KUKA KRL program: EPS_2_251491_MH04A_A_20251118025158.src

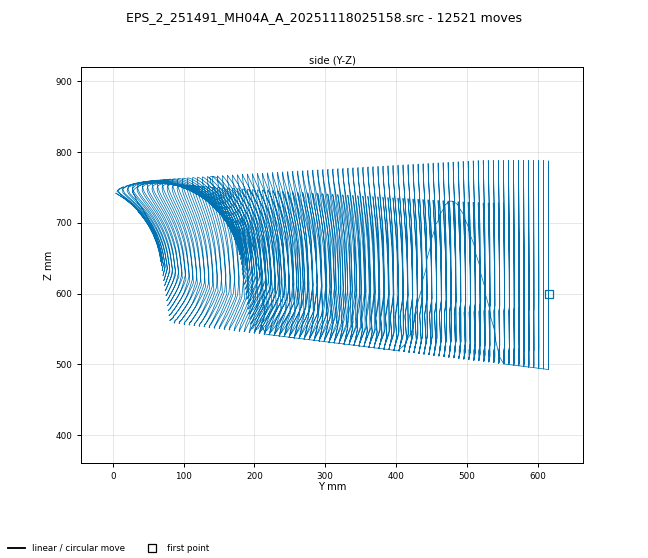
[picture p0: tool path of EPS_2_251491_MH04A_A_20251118025158.src, 12521 of 12523 moves have a stored position in this frame; points joined in program order, loops and branches not executed]
&ACCESS RVP
&REL 4
&COMMENT QRS 19112012
&PARAM EDITMASK = *
DEF PART()
EXT BAS (BAS_COMMAND :IN,REAL :IN )
INT I
BAS (#INITMOV,0 )

;KUKA QRS Post kuka4.cps  Date:22-06-2017 !

File_ID=2918

QRS_PRE_INIT()

;Init var - Until changes are made in qrs_pre_init
Outlet_Square_prg=0
Inlet_1_Square_prg=0
Inlet_2_Square_prg=0
Inlet_3_Square_prg=0
Inlet_4_Square_prg=0
Inlet_5_Square_prg=0

Outlet_1={X 0.000, Y 519.160, Z 687.500, B 0.000, E1 0.000 }
Inlet_1={X 0.000, Y 523.440, Z 627.500, B 0.000, E1 142.000 }
Outlet_1_type=201
Inlet_1_type=201
;QRS#1=Sidecore dimensions
;QRS#2=200-8" PVC SDR 35
;QRS#3=200-8" PVC SDR 35
;QRS#4=
;QRS#5=
;QRS#6=
;QRS#7=
;QRS#8=
;QRS#9=12-08 PSX
;QRS#10=12-08 PSX
;QRS#11=
;QRS#12=
;QRS#13=
;QRS#14=
;QRS#15=
;QRS#16=1220x127x1067 3,5'
;QRS#17=EPS Height
;QRS#18=788
;QRS#19=*
;QRS#20= UPDATED VERSION 22-06-2017
;QRS#21=*
Outlet_Square=0100
Inlet_1_Square=0100
Inlet_2_Square=0
Inlet_3_Square=0
Inlet_4_Square=0
Inlet_5_Square=0
Mill_Square=1
Outlet_Square_Prg=204
Inlet_1_Square_prg=204

QRS_INIT()

$ADVANCE=5

; T1
PTP {E1 173.594,E2 173.594}
PTP {X 0,Y 615.502,A -85,B 0,C 180,E1 173.594,E2 173.594,E3 0,E4 0,E5 0,E6 0}
QRS_SPEED_INIT()
LIN {X 0,Y 615.502,Z 600,A -85,B 0,C 180,E1 173.594,E2 173.594,E3 0,E4 0,E5 0,E6 0} C_VEL
LIN {X 0,Y 615.502,Z 502.864,A -85,B 0,C 180,E1 173.594,E2 173.594} C_VEL
LIN {X 0,Y 615.502,Z 494.687,A -85,B 0,C 180,E1 173.594,E2 173.594} C_VEL
LIN {X 0,Y 615.49,Z 492.687,A -85,B 0,C 180,E1 173.408,E2 173.408} C_VEL
LIN {X 0,Y 615.493,Z 492.697,A -85,B 0,C 180,E1 170.802,E2 170.802} C_VEL
LIN {X 0,Y 615.479,Z 492.685,A -85,B 0,C 180,E1 168.139,E2 168.139} C_VEL
LIN {X 0,Y 615.488,Z 492.686,A -85,B 0,C 180,E1 165.451,E2 165.451} C_VEL
LIN {X 0,Y 615.494,Z 492.696,A -85,B 0,C 180,E1 162.73,E2 162.73} C_VEL
LIN {X 0,Y 615.477,Z 492.684,A -85,B 0,C 180,E1 159.967,E2 159.967} C_VEL
LIN {X 0,Y 615.486,Z 492.692,A -85,B 0,C 180,E1 157.156,E2 157.156} C_VEL
LIN {X 0,Y 615.493,Z 492.685,A -85,B 0,C 180,E1 154.285,E2 154.285} C_VEL
LIN {X 0,Y 615.486,Z 492.686,A -85,B 0,C 180,E1 151.342,E2 151.342} C_VEL
LIN {X 0,Y 615.492,Z 492.697,A -85,B 0,C 180,E1 148.911,E2 148.911} C_VEL
LIN {X 0,Y 615.479,Z 492.684,A -85,B 0,C 180,E1 145.978,E2 145.978} C_VEL
LIN {X 0,Y 615.49,Z 492.767,A -85,B 0,C 180,E1 145.297,E2 145.297} C_VEL
LIN {X 0,Y 615.493,Z 508.915,A -85,B 0,C 180,E1 142.373,E2 142.373} C_VEL
LIN {X 0,Y 615.476,Z 517.644,A -85,B 0,C 180,E1 140.809,E2 140.809} C_VEL
LIN {X 0,Y 615.481,Z 623.163,A -85,B 0,C 180,E1 139.556,E2 139.556} C_VEL
LIN {X 0,Y 615.482,Z 636.415,A -85,B 0,C 180,E1 139.271,E2 139.271} C_VEL
LIN {X 0,Y 615.49,Z 649.214,A -85,B 0,C 180,E1 138.857,E2 138.857} C_VEL
LIN {X 0,Y 615.497,Z 660.234,A -85,B 0,C 180,E1 138.376,E2 138.376} C_VEL
LIN {X 0,Y 615.48,Z 670.961,A -85,B 0,C 180,E1 137.783,E2 137.783} C_VEL
LIN {X 0,Y 615.495,Z 681.65,A -85,B 0,C 180,E1 137.038,E2 137.038} C_VEL
LIN {X 0,Y 615.496,Z 691.498,A -85,B 0,C 180,E1 136.19,E2 136.19} C_VEL
LIN {X 0,Y 615.494,Z 700.206,A -85,B 0,C 180,E1 135.263,E2 135.263} C_VEL
LIN {X 0,Y 615.495,Z 707.231,A -85,B 0,C 180,E1 134.343,E2 134.343} C_VEL
LIN {X 0,Y 615.499,Z 713.951,A -85,B 0,C 180,E1 133.242,E2 133.242} C_VEL
LIN {X 0,Y 615.498,Z 719.396,A -85,B 0,C 180,E1 132.082,E2 132.082} C_VEL
LIN {X 0,Y 615.495,Z 722.82,A -85,B 0,C 180,E1 131.096,E2 131.096} C_VEL
LIN {X 0,Y 615.498,Z 725.29,A -85,B 0,C 180,E1 130.091,E2 130.091} C_VEL
LIN {X 0,Y 615.491,Z 726.968,A -85,B 0,C 180,E1 128.903,E2 128.903} C_VEL
LIN {X 0,Y 615.493,Z 727.381,A -85,B 0,C 180,E1 128.013,E2 128.013} C_VEL
LIN {X 0,Y 615.492,Z 726.916,A -85,B 0,C 180,E1 126.938,E2 126.938} C_VEL
LIN {X 0,Y 615.496,Z 725.326,A -85,B 0,C 180,E1 125.836,E2 125.836} C_VEL
LIN {X 0,Y 615.494,Z 722.463,A -85,B 0,C 180,E1 124.702,E2 124.702} C_VEL
LIN {X 0,Y 615.494,Z 718.151,A -85,B 0,C 180,E1 123.536,E2 123.536} C_VEL
LIN {X 0,Y 615.496,Z 712.793,A -85,B 0,C 180,E1 122.456,E2 122.456} C_VEL
LIN {X 0,Y 615.496,Z 705.972,A -85,B 0,C 180,E1 121.385,E2 121.385} C_VEL
LIN {X 0,Y 615.497,Z 697.582,A -85,B 0,C 180,E1 120.348,E2 120.348} C_VEL
LIN {X 0,Y 615.498,Z 689.18,A -85,B 0,C 180,E1 119.503,E2 119.503} C_VEL
LIN {X 0,Y 615.495,Z 678.79,A -85,B 0,C 180,E1 118.657,E2 118.657} C_VEL
LIN {X 0,Y 615.485,Z 667.368,A -85,B 0,C 180,E1 117.914,E2 117.914} C_VEL
LIN {X 0,Y 615.487,Z 655.583,A -85,B 0,C 180,E1 117.314,E2 117.314} C_VEL
LIN {X 0,Y 615.479,Z 642.588,A -85,B 0,C 180,E1 116.821,E2 116.821} C_VEL
LIN {X 0,Y 615.479,Z 629.925,A -85,B 0,C 180,E1 116.481,E2 116.481} C_VEL
LIN {X 0,Y 615.491,Z 616.108,A -85,B 0,C 180,E1 116.261,E2 116.261} C_VEL
LIN {X 0,Y 615.49,Z 517.628,A -85,B 0,C 180,E1 115.099,E2 115.099} C_VEL
LIN {X 0,Y 615.496,Z 501.148,A -85,B 0,C 180,E1 112.136,E2 112.136} C_VEL
LIN {X 0,Y 615.476,Z 492.688,A -85,B 0,C 180,E1 110.577,E2 110.577} C_VEL
LIN {X 0,Y 615.486,Z 492.683,A -85,B 0,C 180,E1 107.957,E2 107.957} C_VEL
LIN {X 0,Y 615.489,Z 492.699,A -85,B 0,C 180,E1 105.226,E2 105.226} C_VEL
LIN {X 0,Y 615.477,Z 492.688,A -85,B 0,C 180,E1 102.53,E2 102.53} C_VEL
LIN {X 0,Y 615.486,Z 492.683,A -85,B 0,C 180,E1 99.862,E2 99.862} C_VEL
LIN {X 0,Y 615.491,Z 492.698,A -85,B 0,C 180,E1 97.215,E2 97.215} C_VEL
LIN {X 0,Y 615.477,Z 492.689,A -85,B 0,C 180,E1 94.585,E2 94.585} C_VEL
LIN {X 0,Y 615.496,Z 492.68,A -85,B 0,C 180,E1 91.963,E2 91.963} C_VEL
LIN {X 0,Y 615.484,Z 492.694,A -85,B 0,C 180,E1 89.346,E2 89.346} C_VEL
LIN {X 0,Y 615.482,Z 492.692,A -85,B 0,C 180,E1 86.727,E2 86.727} C_VEL
LIN {X 0,Y 615.488,Z 492.681,A -85,B 0,C 180,E1 84.102,E2 84.102} C_VEL
LIN {X 0,Y 615.479,Z 492.691,A -85,B 0,C 180,E1 81.463,E2 81.463} C_VEL
LIN {X 0,Y 615.489,Z 492.694,A -85,B 0,C 180,E1 78.807,E2 78.807} C_VEL
LIN {X 0,Y 615.485,Z 492.682,A -85,B 0,C 180,E1 76.067,E2 76.067} C_VEL
LIN {X 0,Y 615.482,Z 492.691,A -85,B 0,C 180,E1 73.414,E2 73.414} C_VEL
LIN {X 0,Y 615.483,Z 492.691,A -85,B 0,C 180,E1 70.662,E2 70.662} C_VEL
LIN {X 0,Y 615.495,Z 492.68,A -85,B 0,C 180,E1 67.864,E2 67.864} C_VEL
LIN {X 0,Y 615.495,Z 492.701,A -85,B 0,C 180,E1 65.009,E2 65.009} C_VEL
LIN {X 0,Y 615.483,Z 492.683,A -85,B 0,C 180,E1 62.085,E2 62.085} C_VEL
LIN {X 0,Y 615.499,Z 492.679,A -85,B 0,C 180,E1 59.841,E2 59.841} C_VEL
LIN {X 0,Y 615.485,Z 492.686,A -85,B 0,C 180,E1 57.543,E2 57.543} C_VEL
LIN {X 0,Y 615.482,Z 492.696,A -85,B 0,C 180,E1 55.186,E2 55.186} C_VEL
LIN {X 0,Y 615.492,Z 492.694,A -85,B 0,C 180,E1 52.759,E2 52.759} C_VEL
LIN {X 0,Y 615.489,Z 492.681,A -85,B 0,C 180,E1 49.91,E2 49.91} C_VEL
LIN {X 0,Y 615.493,Z 492.701,A -85,B 0,C 180,E1 46.951,E2 46.951} C_VEL
LIN {X 0,Y 615.482,Z 492.683,A -85,B 0,C 180,E1 43.998,E2 43.998} C_VEL
LIN {X 0,Y 615.489,Z 492.696,A -85,B 0,C 180,E1 41.096,E2 41.096} C_VEL
LIN {X 0,Y 615.496,Z 492.7,A -85,B 0,C 180,E1 38.903,E2 38.903} C_VEL
LIN {X 0,Y 615.481,Z 492.689,A -85,B 0,C 180,E1 36.425,E2 36.425} C_VEL
LIN {X 0,Y 615.479,Z 492.684,A -85,B 0,C 180,E1 34.022,E2 34.022} C_VEL
LIN {X 0,Y 615.487,Z 492.683,A -85,B 0,C 180,E1 31.685,E2 31.685} C_VEL
LIN {X 0,Y 615.487,Z 492.687,A -85,B 0,C 180,E1 29.406,E2 29.406} C_VEL
LIN {X 0,Y 615.491,Z 492.696,A -85,B 0,C 180,E1 27.048,E2 27.048} C_VEL
LIN {X 0,Y 615.478,Z 492.687,A -85,B 0,C 180,E1 24.272,E2 24.272} C_VEL
LIN {X 0,Y 615.49,Z 492.685,A -85,B 0,C 180,E1 21.431,E2 21.431} C_VEL
LIN {X 0,Y 615.495,Z 492.692,A -85,B 0,C 180,E1 18.611,E2 18.611} C_VEL
LIN {X 0,Y 615.48,Z 492.683,A -85,B 0,C 180,E1 15.905,E2 15.905} C_VEL
LIN {X 0,Y 615.487,Z 492.69,A -85,B 0,C 180,E1 13.201,E2 13.201} C_VEL
LIN {X 0,Y 615.492,Z 492.691,A -85,B 0,C 180,E1 10.526,E2 10.526} C_VEL
LIN {X 0,Y 615.479,Z 492.684,A -85,B 0,C 180,E1 7.875,E2 7.875} C_VEL
LIN {X 0,Y 615.485,Z 492.689,A -85,B 0,C 180,E1 5.241,E2 5.241} C_VEL
LIN {X 0,Y 615.497,Z 492.694,A -85,B 0,C 180,E1 2.617,E2 2.617} C_VEL
LIN {X 0,Y 615.477,Z 492.685,A -85,B 0,C 180,E1 0,E2 0} C_VEL
LIN {X 0,Y 615.494,Z 492.684,A -85,B 0,C 180,E1 -2.618,E2 -2.618} C_VEL
LIN {X 0,Y 615.496,Z 492.7,A -85,B 0,C 180,E1 -5.241,E2 -5.241} C_VEL
LIN {X 0,Y 615.479,Z 492.686,A -85,B 0,C 180,E1 -7.876,E2 -7.876} C_VEL
LIN {X 0,Y 615.49,Z 492.683,A -85,B 0,C 180,E1 -10.527,E2 -10.527} C_VEL
LIN {X 0,Y 615.497,Z 492.699,A -85,B 0,C 180,E1 -13.201,E2 -13.201} C_VEL
LIN {X 0,Y 615.48,Z 492.686,A -85,B 0,C 180,E1 -15.906,E2 -15.906} C_VEL
LIN {X 0,Y 615.491,Z 492.684,A -85,B 0,C 180,E1 -18.646,E2 -18.646} C_VEL
LIN {X 0,Y 615.497,Z 492.695,A -85,B 0,C 180,E1 -21.432,E2 -21.432} C_VEL
LIN {X 0,Y 615.478,Z 492.684,A -85,B 0,C 180,E1 -24.273,E2 -24.273} C_VEL
LIN {X 0,Y 615.491,Z 492.693,A -85,B 0,C 180,E1 -27.048,E2 -27.048} C_VEL
LIN {X 0,Y 615.488,Z 492.687,A -85,B 0,C 180,E1 -29.797,E2 -29.797} C_VEL
LIN {X 0,Y 615.484,Z 492.683,A -85,B 0,C 180,E1 -32.458,E2 -32.458} C_VEL
LIN {X 0,Y 615.494,Z 492.685,A -85,B 0,C 180,E1 -34.815,E2 -34.815} C_VEL
LIN {X 0,Y 615.49,Z 492.699,A -85,B 0,C 180,E1 -37.242,E2 -37.242} C_VEL
LIN {X 0,Y 615.478,Z 492.685,A -85,B 0,C 180,E1 -40.09,E2 -40.09} C_VEL
LIN {X 0,Y 615.478,Z 492.684,A -85,B 0,C 180,E1 -42.354,E2 -42.354} C_VEL
LIN {X 0,Y 615.49,Z 492.692,A -85,B 0,C 180,E1 -45.069,E2 -45.069} C_VEL
LIN {X 0,Y 615.488,Z 492.686,A -85,B 0,C 180,E1 -47.92,E2 -47.92} C_VEL
LIN {X 0,Y 615.477,Z 492.684,A -85,B 0,C 180,E1 -50.25,E2 -50.25} C_VEL
LIN {X 0,Y 615.492,Z 492.691,A -85,B 0,C 180,E1 -53.063,E2 -53.063} C_VEL
LIN {X 0,Y 615.487,Z 492.685,A -85,B 0,C 180,E1 -55.979,E2 -55.979} C_VEL
LIN {X 0,Y 615.492,Z 492.686,A -85,B 0,C 180,E1 -58.914,E2 -58.914} C_VEL
LIN {X 0,Y 615.482,Z 492.698,A -85,B 0,C 180,E1 -61.551,E2 -61.551} C_VEL
LIN {X 0,Y 615.477,Z 492.684,A -85,B 0,C 180,E1 -64.284,E2 -64.284} C_VEL
LIN {X 0,Y 615.482,Z 492.877,A -85,B 0,C 180,E1 -66.711,E2 -66.711} C_VEL
LIN {X 0,Y 615.476,Z 514.047,A -85,B 0,C 180,E1 -69.447,E2 -69.447} C_VEL
LIN {X 0,Y 615.48,Z 535.84,A -85,B 0,C 180,E1 -72.215,E2 -72.215} C_VEL
LIN {X 0,Y 615.492,Z 557.627,A -85,B 0,C 180,E1 -74.944,E2 -74.944} C_VEL
LIN {X 0,Y 615.488,Z 575.134,A -85,B 0,C 180,E1 -77.114,E2 -77.114} C_VEL
LIN {X 0,Y 615.477,Z 683.848,A -85,B 0,C 180,E1 -78.411,E2 -78.411} C_VEL
LIN {X 0,Y 615.482,Z 696.355,A -85,B 0,C 180,E1 -78.682,E2 -78.682} C_VEL
LIN {X 0,Y 615.497,Z 709.491,A -85,B 0,C 180,E1 -79.109,E2 -79.109} C_VEL
LIN {X 0,Y 615.48,Z 721.483,A -85,B 0,C 180,E1 -79.64,E2 -79.64} C_VEL
LIN {X 0,Y 615.481,Z 733,A -85,B 0,C 180,E1 -80.304,E2 -80.304} C_VEL
LIN {X 0,Y 615.499,Z 743.344,A -85,B 0,C 180,E1 -81.05,E2 -81.05} C_VEL
LIN {X 0,Y 615.497,Z 751.814,A -85,B 0,C 180,E1 -81.794,E2 -81.794} C_VEL
LIN {X 0,Y 615.498,Z 759.608,A -85,B 0,C 180,E1 -82.62,E2 -82.62} C_VEL
LIN {X 0,Y 615.496,Z 767.204,A -85,B 0,C 180,E1 -83.608,E2 -83.608} C_VEL
LIN {X 0,Y 615.498,Z 774.205,A -85,B 0,C 180,E1 -84.759,E2 -84.759} C_VEL
LIN {X 0,Y 615.493,Z 778.852,A -85,B 0,C 180,E1 -85.744,E2 -85.744} C_VEL
LIN {X 0,Y 615.495,Z 782.399,A -85,B 0,C 180,E1 -86.727,E2 -86.727} C_VEL
LIN {X 0,Y 615.497,Z 784.233,A -85,B 0,C 180,E1 -87.382,E2 -87.382} C_VEL
LIN {X 0,Y 615.496,Z 785.608,A -85,B 0,C 180,E1 -88.037,E2 -88.037} C_VEL
LIN {X 0,Y 615.496,Z 787.174,A -85,B 0,C 180,E1 -89.346,E2 -89.346} C_VEL
LIN {X 0,Y 615.494,Z 787.389,A -85,B 0,C 180,E1 -90,E2 -90} C_VEL
LIN {X 0,Y 615.496,Z 786.58,A -85,B 0,C 180,E1 -91.309,E2 -91.309} C_VEL
LIN {X 0,Y 615.496,Z 785.608,A -85,B 0,C 180,E1 -91.963,E2 -91.963} C_VEL
LIN {X 0,Y 615.497,Z 784.233,A -85,B 0,C 180,E1 -92.618,E2 -92.618} C_VEL
LIN {X 0,Y 615.496,Z 781.35,A -85,B 0,C 180,E1 -93.601,E2 -93.601} C_VEL
LIN {X 0,Y 615.498,Z 777.442,A -85,B 0,C 180,E1 -94.584,E2 -94.584} C_VEL
LIN {X 0,Y 615.499,Z 772.406,A -85,B 0,C 180,E1 -95.57,E2 -95.57} C_VEL
LIN {X 0,Y 615.497,Z 765.87,A -85,B 0,C 180,E1 -96.583,E2 -96.583} C_VEL
LIN {X 0,Y 615.497,Z 758.135,A -85,B 0,C 180,E1 -97.545,E2 -97.545} C_VEL
LIN {X 0,Y 615.498,Z 750.047,A -85,B 0,C 180,E1 -98.371,E2 -98.371} C_VEL
LIN {X 0,Y 615.499,Z 740.17,A -85,B 0,C 180,E1 -99.198,E2 -99.198} C_VEL
LIN {X 0,Y 615.483,Z 728.986,A -85,B 0,C 180,E1 -99.945,E2 -99.945} C_VEL
LIN {X 0,Y 615.481,Z 718.029,A -85,B 0,C 180,E1 -100.527,E2 -100.527} C_VEL
LIN {X 0,Y 615.499,Z 705.424,A -85,B 0,C 180,E1 -101.042,E2 -101.042} C_VEL
LIN {X 0,Y 615.479,Z 693.079,A -85,B 0,C 180,E1 -101.401,E2 -101.401} C_VEL
LIN {X 0,Y 615.477,Z 679.489,A -85,B 0,C 180,E1 -101.652,E2 -101.652} C_VEL
LIN {X 0,Y 615.488,Z 575.134,A -85,B 0,C 180,E1 -102.886,E2 -102.886} C_VEL
LIN {X 0,Y 615.479,Z 552.18,A -85,B 0,C 180,E1 -105.735,E2 -105.735} C_VEL
LIN {X 0,Y 615.481,Z 530.652,A -85,B 0,C 180,E1 -108.44,E2 -108.44} C_VEL
LIN {X 0,Y 615.488,Z 508.571,A -85,B 0,C 180,E1 -111.256,E2 -111.256} C_VEL
LIN {X 0,Y 615.484,Z 492.684,A -85,B 0,C 180,E1 -113.333,E2 -113.333} C_VEL
LIN {X 0,Y 615.477,Z 492.684,A -85,B 0,C 180,E1 -115.716,E2 -115.716} C_VEL
LIN {X 0,Y 615.482,Z 492.698,A -85,B 0,C 180,E1 -118.449,E2 -118.449} C_VEL
LIN {X 0,Y 615.493,Z 492.687,A -85,B 0,C 180,E1 -121.086,E2 -121.086} C_VEL
LIN {X 0,Y 615.487,Z 492.685,A -85,B 0,C 180,E1 -124.021,E2 -124.021} C_VEL
LIN {X 0,Y 615.492,Z 492.692,A -85,B 0,C 180,E1 -126.937,E2 -126.937} C_VEL
LIN {X 0,Y 615.477,Z 492.684,A -85,B 0,C 180,E1 -129.75,E2 -129.75} C_VEL
LIN {X 0,Y 615.49,Z 492.69,A -85,B 0,C 180,E1 -132.351,E2 -132.351} C_VEL
LIN {X 0,Y 615.489,Z 492.69,A -85,B 0,C 180,E1 -135.067,E2 -135.067} C_VEL
LIN {X 0,Y 615.477,Z 492.684,A -85,B 0,C 180,E1 -137.646,E2 -137.646} C_VEL
LIN {X 0,Y 615.498,Z 492.684,A -85,B 0,C 180,E1 -140.25,E2 -140.25} C_VEL
LIN {X 0,Y 615.491,Z 492.692,A -85,B 0,C 180,E1 -143.061,E2 -143.061} C_VEL
LIN {X 0,Y 615.493,Z 492.686,A -85,B 0,C 180,E1 -145.297,E2 -145.297} C_VEL
LIN {X 0,Y 615.479,Z 492.684,A -85,B 0,C 180,E1 -147.668,E2 -147.668} C_VEL
LIN {X 0,Y 615.488,Z 492.685,A -85,B 0,C 180,E1 -150.203,E2 -150.203} C_VEL
LIN {X 0,Y 615.496,Z 492.697,A -85,B 0,C 180,E1 -152.951,E2 -152.951} C_VEL
LIN {X 0,Y 615.478,Z 492.684,A -85,B 0,C 180,E1 -155.727,E2 -155.727} C_VEL
LIN {X 0,Y 615.477,Z 492.684,A -85,B 0,C 180,E1 -157.863,E2 -157.863} C_VEL
LIN {X 0,Y 615.486,Z 492.695,A -85,B 0,C 180,E1 -160.662,E2 -160.662} C_VEL
LIN {X 0,Y 615.485,Z 492.685,A -85,B 0,C 180,E1 -163.565,E2 -163.565} C_VEL
LIN {X 0,Y 615.476,Z 492.685,A -85,B 0,C 180,E1 -166.125,E2 -166.125} C_VEL
LIN {X 0,Y 615.485,Z 492.698,A -85,B 0,C 180,E1 -168.807,E2 -168.807} C_VEL
LIN {X 0,Y 615.492,Z 492.686,A -85,B 0,C 180,E1 -171.463,E2 -171.463} C_VEL
LIN {X 0,Y 615.478,Z 492.684,A -85,B 0,C 180,E1 -174.101,E2 -174.101} C_VEL
LIN {X 0,Y 615.484,Z 492.694,A -85,B 0,C 180,E1 -176.727,E2 -176.727} C_VEL
LIN {X 0,Y 615.493,Z 492.69,A -85,B 0,C 180,E1 -179.345,E2 -179.345} C_VEL
LIN {X 0,Y 615.477,Z 492.684,A -85,B 0,C 180,E1 -181.963,E2 -181.963} C_VEL
LIN {X 0,Y 615.495,Z 492.686,A -85,B 0,C 180,E1 -184.584,E2 -184.584} C_VEL
LIN {X 0,Y 615.49,Z 492.687,A -85,B 0,C 180,E1 -186.592,E2 -186.592} C_VEL
LIN {X 0,Y 614.816,Z 492.842,A -85,B 0,C 180,E1 -187.138,E2 -187.138} C_VEL
LIN {X 0,Y 611.984,Z 493.247,A -85,B 0,C 180,E1 -188.024,E2 -188.024} C_VEL
LIN {X 0,Y 609.59,Z 493.561,A -85,B 0,C 180,E1 -188.736,E2 -188.736} C_VEL
LIN {X 0,Y 608.551,Z 493.682,A -85,B 0,C 180,E1 -189.286,E2 -189.286} C_VEL
LIN {X 0,Y 608.459,Z 493.69,A -85,B 0,C 180,E1 -189.472,E2 -189.472} C_VEL
LIN {X 0,Y 608.456,Z 493.686,A -85,B 0,C 180,E1 -192,E2 -192} C_VEL
LIN {X 0,Y 608.476,Z 493.688,A -85,B 0,C 180,E1 -194.72,E2 -194.72} C_VEL
LIN {X 0,Y 608.454,Z 493.692,A -85,B 0,C 180,E1 -197.476,E2 -197.476} C_VEL
LIN {X 0,Y 608.458,Z 493.686,A -85,B 0,C 180,E1 -200.274,E2 -200.274} C_VEL
LIN {X 0,Y 608.45,Z 493.688,A -85,B 0,C 180,E1 -202.477,E2 -202.477} C_VEL
LIN {X 0,Y 608.455,Z 493.696,A -85,B 0,C 180,E1 -205.3,E2 -205.3} C_VEL
LIN {X 0,Y 608.446,Z 493.693,A -85,B 0,C 180,E1 -207.518,E2 -207.518} C_VEL
LIN {X 0,Y 608.464,Z 493.686,A -85,B 0,C 180,E1 -209.973,E2 -209.973} C_VEL
LIN {X 0,Y 608.458,Z 493.687,A -85,B 0,C 180,E1 -212.524,E2 -212.524} C_VEL
LIN {X 0,Y 608.493,Z 493.764,A -85,B 0,C 180,E1 -214.661,E2 -214.661} C_VEL
LIN {X 0,Y 608.466,Z 508.89,A -85,B 0,C 180,E1 -217.421,E2 -217.421} C_VEL
LIN {X 0,Y 608.461,Z 517.864,A -85,B 0,C 180,E1 -219.042,E2 -219.042} C_VEL
LIN {X 0,Y 608.543,Z 623.86,A -85,B 0,C 180,E1 -220.32,E2 -220.32} C_VEL
LIN {X 0,Y 608.53,Z 637.415,A -85,B 0,C 180,E1 -220.622,E2 -220.622} C_VEL
LIN {X 0,Y 608.537,Z 650.476,A -85,B 0,C 180,E1 -221.059,E2 -221.059} C_VEL
LIN {X 0,Y 608.503,Z 661.811,A -85,B 0,C 180,E1 -221.573,E2 -221.573} C_VEL
LIN {X 0,Y 608.48,Z 673.814,A -85,B 0,C 180,E1 -222.277,E2 -222.277} C_VEL
LIN {X 0,Y 608.478,Z 684.29,A -85,B 0,C 180,E1 -223.046,E2 -223.046} C_VEL
LIN {X 0,Y 608.484,Z 693.364,A -85,B 0,C 180,E1 -223.868,E2 -223.868} C_VEL
LIN {X 0,Y 608.468,Z 701.727,A -85,B 0,C 180,E1 -224.794,E2 -224.794} C_VEL
LIN {X 0,Y 608.449,Z 708.679,A -85,B 0,C 180,E1 -225.736,E2 -225.736} C_VEL
LIN {X 0,Y 608.436,Z 714.414,A -85,B 0,C 180,E1 -226.694,E2 -226.694} C_VEL
LIN {X 0,Y 608.437,Z 719.065,A -85,B 0,C 180,E1 -227.668,E2 -227.668} C_VEL
LIN {X 0,Y 608.431,Z 723.238,A -85,B 0,C 180,E1 -228.823,E2 -228.823} C_VEL
LIN {X 0,Y 608.444,Z 725.473,A -85,B 0,C 180,E1 -229.697,E2 -229.697} C_VEL
LIN {X 0,Y 608.42,Z 727.168,A -85,B 0,C 180,E1 -230.708,E2 -230.708} C_VEL
LIN {X 0,Y 608.414,Z 727.941,A -85,B 0,C 180,E1 -231.765,E2 -231.765} C_VEL
LIN {X 0,Y 608.429,Z 727.512,A -85,B 0,C 180,E1 -233.084,E2 -233.084} C_VEL
LIN {X 0,Y 608.419,Z 726.323,A -85,B 0,C 180,E1 -233.957,E2 -233.957} C_VEL
LIN {X 0,Y 608.42,Z 723.731,A -85,B 0,C 180,E1 -235.098,E2 -235.098} C_VEL
LIN {X 0,Y 608.455,Z 719.461,A -85,B 0,C 180,E1 -236.33,E2 -236.33} C_VEL
LIN {X 0,Y 608.434,Z 713.949,A -85,B 0,C 180,E1 -237.481,E2 -237.481} C_VEL
LIN {X 0,Y 608.457,Z 707.761,A -85,B 0,C 180,E1 -238.49,E2 -238.49} C_VEL
LIN {X 0,Y 608.455,Z 700.429,A -85,B 0,C 180,E1 -239.455,E2 -239.455} C_VEL
LIN {X 0,Y 608.461,Z 691.422,A -85,B 0,C 180,E1 -240.411,E2 -240.411} C_VEL
LIN {X 0,Y 608.496,Z 682.113,A -85,B 0,C 180,E1 -241.216,E2 -241.216} C_VEL
LIN {X 0,Y 608.507,Z 672.117,A -85,B 0,C 180,E1 -241.925,E2 -241.925} C_VEL
LIN {X 0,Y 608.504,Z 660.528,A -85,B 0,C 180,E1 -242.581,E2 -242.581} C_VEL
LIN {X 0,Y 608.51,Z 648.245,A -85,B 0,C 180,E1 -243.115,E2 -243.115} C_VEL
LIN {X 0,Y 608.531,Z 635.132,A -85,B 0,C 180,E1 -243.531,E2 -243.531} C_VEL
LIN {X 0,Y 608.56,Z 622.833,A -85,B 0,C 180,E1 -243.786,E2 -243.786} C_VEL
LIN {X 0,Y 608.458,Z 517.892,A -85,B 0,C 180,E1 -245.043,E2 -245.043} C_VEL
LIN {X 0,Y 608.489,Z 501.824,A -85,B 0,C 180,E1 -247.953,E2 -247.953} C_VEL
LIN {X 0,Y 608.459,Z 493.688,A -85,B 0,C 180,E1 -249.467,E2 -249.467} C_VEL
LIN {X 0,Y 608.446,Z 493.688,A -85,B 0,C 180,E1 -251.829,E2 -251.829} C_VEL
LIN {X 0,Y 608.473,Z 493.691,A -85,B 0,C 180,E1 -254.594,E2 -254.594} C_VEL
LIN {X 0,Y 608.469,Z 493.688,A -85,B 0,C 180,E1 -257.323,E2 -257.323} C_VEL
LIN {X 0,Y 608.454,Z 493.687,A -85,B 0,C 180,E1 -260.023,E2 -260.023} C_VEL
LIN {X 0,Y 608.485,Z 493.69,A -85,B 0,C 180,E1 -262.701,E2 -262.701} C_VEL
LIN {X 0,Y 608.447,Z 493.691,A -85,B 0,C 180,E1 -265.362,E2 -265.362} C_VEL
LIN {X 0,Y 608.466,Z 493.685,A -85,B 0,C 180,E1 -268.014,E2 -268.014} C_VEL
LIN {X 0,Y 608.478,Z 493.69,A -85,B 0,C 180,E1 -270.662,E2 -270.662} C_VEL
LIN {X 0,Y 608.476,Z 493.688,A -85,B 0,C 180,E1 -273.311,E2 -273.311} C_VEL
LIN {X 0,Y 608.484,Z 493.683,A -85,B 0,C 180,E1 -275.967,E2 -275.967} C_VEL
LIN {X 0,Y 608.451,Z 493.693,A -85,B 0,C 180,E1 -278.636,E2 -278.636} C_VEL
LIN {X 0,Y 608.478,Z 493.688,A -85,B 0,C 180,E1 -281.323,E2 -281.323} C_VEL
LIN {X 0,Y 608.466,Z 493.685,A -85,B 0,C 180,E1 -284.037,E2 -284.037} C_VEL
LIN {X 0,Y 608.472,Z 493.692,A -85,B 0,C 180,E1 -286.783,E2 -286.783} C_VEL
LIN {X 0,Y 608.452,Z 493.689,A -85,B 0,C 180,E1 -289.57,E2 -289.57} C_VEL
LIN {X 0,Y 608.454,Z 493.689,A -85,B 0,C 180,E1 -292.476,E2 -292.476} C_VEL
LIN {X 0,Y 608.457,Z 493.69,A -85,B 0,C 180,E1 -294.57,E2 -294.57} C_VEL
LIN {X 0,Y 608.484,Z 493.69,A -85,B 0,C 180,E1 -297.209,E2 -297.209} C_VEL
LIN {X 0,Y 608.465,Z 493.685,A -85,B 0,C 180,E1 -299.972,E2 -299.972} C_VEL
LIN {X 0,Y 608.46,Z 493.689,A -85,B 0,C 180,E1 -302.523,E2 -302.523} C_VEL
LIN {X 0,Y 608.436,Z 493.696,A -85,B 0,C 180,E1 -305.277,E2 -305.277} C_VEL
LIN {X 0,Y 608.47,Z 493.686,A -85,B 0,C 180,E1 -307.745,E2 -307.745} C_VEL
LIN {X 0,Y 608.474,Z 493.685,A -85,B 0,C 180,E1 -310.332,E2 -310.332} C_VEL
LIN {X 0,Y 608.484,Z 493.689,A -85,B 0,C 180,E1 -313.311,E2 -313.311} C_VEL
LIN {X 0,Y 608.467,Z 493.685,A -85,B 0,C 180,E1 -316.131,E2 -316.131} C_VEL
LIN {X 0,Y 608.458,Z 493.693,A -85,B 0,C 180,E1 -318.824,E2 -318.824} C_VEL
LIN {X 0,Y 608.471,Z 493.69,A -85,B 0,C 180,E1 -321.413,E2 -321.413} C_VEL
LIN {X 0,Y 608.469,Z 493.685,A -85,B 0,C 180,E1 -323.95,E2 -323.95} C_VEL
LIN {X 0,Y 608.463,Z 493.686,A -85,B 0,C 180,E1 -326.33,E2 -326.33} C_VEL
LIN {X 0,Y 608.471,Z 493.689,A -85,B 0,C 180,E1 -328.726,E2 -328.726} C_VEL
LIN {X 0,Y 608.473,Z 493.691,A -85,B 0,C 180,E1 -331.378,E2 -331.378} C_VEL
LIN {X 0,Y 608.475,Z 493.684,A -85,B 0,C 180,E1 -334.276,E2 -334.276} C_VEL
LIN {X 0,Y 608.454,Z 493.693,A -85,B 0,C 180,E1 -336.877,E2 -336.877} C_VEL
LIN {X 0,Y 608.459,Z 493.688,A -85,B 0,C 180,E1 -339.726,E2 -339.726} C_VEL
LIN {X 0,Y 608.45,Z 493.689,A -85,B 0,C 180,E1 -342.524,E2 -342.524} C_VEL
LIN {X 0,Y 608.476,Z 493.693,A -85,B 0,C 180,E1 -345.28,E2 -345.28} C_VEL
LIN {X 0,Y 608.457,Z 493.687,A -85,B 0,C 180,E1 -348,E2 -348} C_VEL
LIN {X 0,Y 608.469,Z 493.688,A -85,B 0,C 180,E1 -350.695,E2 -350.695} C_VEL
LIN {X 0,Y 608.465,Z 493.693,A -85,B 0,C 180,E1 -353.368,E2 -353.368} C_VEL
LIN {X 0,Y 608.446,Z 493.688,A -85,B 0,C 180,E1 -356.026,E2 -356.026} C_VEL
LIN {X 0,Y 608.472,Z 493.687,A -85,B 0,C 180,E1 -358.677,E2 -358.677} C_VEL
LIN {X 0,Y 608.477,Z 493.693,A -85,B 0,C 180,E1 -361.324,E2 -361.324} C_VEL
LIN {X 0,Y 608.445,Z 493.689,A -85,B 0,C 180,E1 -363.974,E2 -363.974} C_VEL
LIN {X 0,Y 608.466,Z 493.687,A -85,B 0,C 180,E1 -366.633,E2 -366.633} C_VEL
LIN {X 0,Y 608.476,Z 493.694,A -85,B 0,C 180,E1 -369.306,E2 -369.306} C_VEL
LIN {X 0,Y 608.457,Z 493.687,A -85,B 0,C 180,E1 -372,E2 -372} C_VEL
LIN {X 0,Y 608.477,Z 493.686,A -85,B 0,C 180,E1 -374.721,E2 -374.721} C_VEL
LIN {X 0,Y 608.457,Z 493.693,A -85,B 0,C 180,E1 -377.477,E2 -377.477} C_VEL
LIN {X 0,Y 608.458,Z 493.686,A -85,B 0,C 180,E1 -380.275,E2 -380.275} C_VEL
LIN {X 0,Y 608.451,Z 493.688,A -85,B 0,C 180,E1 -382.478,E2 -382.478} C_VEL
LIN {X 0,Y 608.454,Z 493.698,A -85,B 0,C 180,E1 -385.301,E2 -385.301} C_VEL
LIN {X 0,Y 608.447,Z 493.694,A -85,B 0,C 180,E1 -387.518,E2 -387.518} C_VEL
LIN {X 0,Y 608.464,Z 493.687,A -85,B 0,C 180,E1 -389.973,E2 -389.973} C_VEL
LIN {X 0,Y 608.458,Z 493.687,A -85,B 0,C 180,E1 -392.524,E2 -392.524} C_VEL
LIN {X 0,Y 608.452,Z 493.698,A -85,B 0,C 180,E1 -395.277,E2 -395.277} C_VEL
LIN {X 0,Y 608.467,Z 493.689,A -85,B 0,C 180,E1 -397.747,E2 -397.747} C_VEL
LIN {X 0,Y 608.447,Z 493.688,A -85,B 0,C 180,E1 -400.33,E2 -400.33} C_VEL
LIN {X 0,Y 608.48,Z 493.694,A -85,B 0,C 180,E1 -403.311,E2 -403.311} C_VEL
LIN {X 0,Y 608.469,Z 493.685,A -85,B 0,C 180,E1 -406.132,E2 -406.132} C_VEL
LIN {X 0,Y 608.458,Z 493.689,A -85,B 0,C 180,E1 -408.825,E2 -408.825} C_VEL
LIN {X 0,Y 608.47,Z 493.689,A -85,B 0,C 180,E1 -411.76,E2 -411.76} C_VEL
LIN {X 0,Y 608.474,Z 493.686,A -85,B 0,C 180,E1 -413.951,E2 -413.951} C_VEL
LIN {X 0,Y 608.464,Z 493.686,A -85,B 0,C 180,E1 -416.33,E2 -416.33} C_VEL
LIN {X 0,Y 608.478,Z 493.685,A -85,B 0,C 180,E1 -418.728,E2 -418.728} C_VEL
LIN {X 0,Y 608.472,Z 493.696,A -85,B 0,C 180,E1 -421.381,E2 -421.381} C_VEL
LIN {X 0,Y 608.439,Z 493.691,A -85,B 0,C 180,E1 -423.965,E2 -423.965} C_VEL
LIN {X 0,Y 608.454,Z 493.73,A -85,B 0,C 180,E1 -426.539,E2 -426.539} C_VEL
LIN {X 0,Y 608.581,Z 507.207,A -85,B 0,C 180,E1 -428.313,E2 -428.313} C_VEL
LIN {X 0,Y 608.544,Z 527.677,A -85,B 0,C 180,E1 -430.959,E2 -430.959} C_VEL
LIN {X 0,Y 608.501,Z 549.578,A -85,B 0,C 180,E1 -433.744,E2 -433.744} C_VEL
LIN {X 0,Y 608.478,Z 572.713,A -85,B 0,C 180,E1 -436.644,E2 -436.644} C_VEL
LIN {X 0,Y 608.499,Z 575.357,A -85,B 0,C 180,E1 -436.974,E2 -436.974} C_VEL
LIN {X 0,Y 608.534,Z 683.962,A -85,B 0,C 180,E1 -438.277,E2 -438.277} C_VEL
LIN {X 0,Y 608.533,Z 697.226,A -85,B 0,C 180,E1 -438.572,E2 -438.572} C_VEL
LIN {X 0,Y 608.544,Z 710.336,A -85,B 0,C 180,E1 -439.009,E2 -439.009} C_VEL
LIN {X 0,Y 608.498,Z 721.64,A -85,B 0,C 180,E1 -439.519,E2 -439.519} C_VEL
LIN {X 0,Y 608.471,Z 733.201,A -85,B 0,C 180,E1 -440.191,E2 -440.191} C_VEL
LIN {X 0,Y 608.485,Z 743.596,A -85,B 0,C 180,E1 -440.946,E2 -440.946} C_VEL
LIN {X 0,Y 608.475,Z 752.114,A -85,B 0,C 180,E1 -441.699,E2 -441.699} C_VEL
LIN {X 0,Y 608.471,Z 759.962,A -85,B 0,C 180,E1 -442.534,E2 -442.534} C_VEL
LIN {X 0,Y 608.461,Z 767.287,A -85,B 0,C 180,E1 -443.485,E2 -443.485} C_VEL
LIN {X 0,Y 608.45,Z 772.867,A -85,B 0,C 180,E1 -444.366,E2 -444.366} C_VEL
LIN {X 0,Y 608.432,Z 777.951,A -85,B 0,C 180,E1 -445.362,E2 -445.362} C_VEL
LIN {X 0,Y 608.449,Z 781.896,A -85,B 0,C 180,E1 -446.358,E2 -446.358} C_VEL
LIN {X 0,Y 608.425,Z 784.809,A -85,B 0,C 180,E1 -447.352,E2 -447.352} C_VEL
LIN {X 0,Y 608.441,Z 786.201,A -85,B 0,C 180,E1 -448.014,E2 -448.014} C_VEL
LIN {X 0,Y 608.438,Z 787.783,A -85,B 0,C 180,E1 -449.338,E2 -449.338} C_VEL
LIN {X 0,Y 608.434,Z 788,A -85,B 0,C 180,E1 -450,E2 -450} C_VEL
LIN {X 0,Y 608.448,Z 787.184,A -85,B 0,C 180,E1 -451.324,E2 -451.324} C_VEL
LIN {X 0,Y 608.441,Z 786.201,A -85,B 0,C 180,E1 -451.986,E2 -451.986} C_VEL
LIN {X 0,Y 608.425,Z 784.809,A -85,B 0,C 180,E1 -452.648,E2 -452.648} C_VEL
LIN {X 0,Y 608.449,Z 781.896,A -85,B 0,C 180,E1 -453.642,E2 -453.642} C_VEL
LIN {X 0,Y 608.432,Z 777.951,A -85,B 0,C 180,E1 -454.638,E2 -454.638} C_VEL
LIN {X 0,Y 608.437,Z 771.877,A -85,B 0,C 180,E1 -455.801,E2 -455.801} C_VEL
LIN {X 0,Y 608.462,Z 765.236,A -85,B 0,C 180,E1 -456.799,E2 -456.799} C_VEL
LIN {X 0,Y 608.456,Z 756.991,A -85,B 0,C 180,E1 -457.8,E2 -457.8} C_VEL
LIN {X 0,Y 608.472,Z 748.539,A -85,B 0,C 180,E1 -458.636,E2 -458.636} C_VEL
LIN {X 0,Y 608.474,Z 738.094,A -85,B 0,C 180,E1 -459.473,E2 -459.473} C_VEL
LIN {X 0,Y 608.482,Z 727.76,A -85,B 0,C 180,E1 -460.145,E2 -460.145} C_VEL
LIN {X 0,Y 608.521,Z 716.245,A -85,B 0,C 180,E1 -460.741,E2 -460.741} C_VEL
LIN {X 0,Y 608.528,Z 704.883,A -85,B 0,C 180,E1 -461.192,E2 -461.192} C_VEL
LIN {X 0,Y 608.524,Z 691.365,A -85,B 0,C 180,E1 -461.576,E2 -461.576} C_VEL
LIN {X 0,Y 608.544,Z 678.106,A -85,B 0,C 180,E1 -461.808,E2 -461.808} C_VEL
LIN {X 0,Y 608.489,Z 575.272,A -85,B 0,C 180,E1 -463.037,E2 -463.037} C_VEL
LIN {X 0,Y 608.488,Z 553.607,A -85,B 0,C 180,E1 -465.749,E2 -465.749} C_VEL
LIN {X 0,Y 608.545,Z 531.948,A -85,B 0,C 180,E1 -468.494,E2 -468.494} C_VEL
LIN {X 0,Y 608.596,Z 511.301,A -85,B 0,C 180,E1 -471.153,E2 -471.153} C_VEL
LIN {X 0,Y 608.513,Z 493.901,A -85,B 0,C 180,E1 -473.436,E2 -473.436} C_VEL
LIN {X 0,Y 608.466,Z 493.688,A -85,B 0,C 180,E1 -473.844,E2 -473.844} C_VEL
LIN {X 0,Y 608.454,Z 493.695,A -85,B 0,C 180,E1 -476.773,E2 -476.773} C_VEL
LIN {X 0,Y 608.468,Z 493.689,A -85,B 0,C 180,E1 -479.019,E2 -479.019} C_VEL
LIN {X 0,Y 608.477,Z 493.685,A -85,B 0,C 180,E1 -481.315,E2 -481.315} C_VEL
LIN {X 0,Y 608.471,Z 493.685,A -85,B 0,C 180,E1 -483.734,E2 -483.734} C_VEL
LIN {X 0,Y 608.475,Z 493.686,A -85,B 0,C 180,E1 -486.089,E2 -486.089} C_VEL
LIN {X 0,Y 608.472,Z 493.694,A -85,B 0,C 180,E1 -488.587,E2 -488.587} C_VEL
LIN {X 0,Y 608.462,Z 493.687,A -85,B 0,C 180,E1 -491.342,E2 -491.342} C_VEL
LIN {X 0,Y 608.46,Z 493.689,A -85,B 0,C 180,E1 -494.264,E2 -494.264} C_VEL
LIN {X 0,Y 608.458,Z 493.692,A -85,B 0,C 180,E1 -497.04,E2 -497.04} C_VEL
LIN {X 0,Y 608.446,Z 493.688,A -85,B 0,C 180,E1 -499.696,E2 -499.696} C_VEL
LIN {X 0,Y 608.467,Z 493.688,A -85,B 0,C 180,E1 -502.253,E2 -502.253} C_VEL
LIN {X 0,Y 608.484,Z 493.689,A -85,B 0,C 180,E1 -505.088,E2 -505.088} C_VEL
LIN {X 0,Y 608.462,Z 493.686,A -85,B 0,C 180,E1 -507.905,E2 -507.905} C_VEL
LIN {X 0,Y 608.472,Z 493.686,A -85,B 0,C 180,E1 -510.22,E2 -510.22} C_VEL
LIN {X 0,Y 608.481,Z 493.694,A -85,B 0,C 180,E1 -512.79,E2 -512.79} C_VEL
LIN {X 0,Y 608.451,Z 493.689,A -85,B 0,C 180,E1 -515.429,E2 -515.429} C_VEL
LIN {X 0,Y 608.463,Z 493.688,A -85,B 0,C 180,E1 -518.308,E2 -518.308} C_VEL
LIN {X 0,Y 608.472,Z 493.689,A -85,B 0,C 180,E1 -521.28,E2 -521.28} C_VEL
LIN {X 0,Y 608.456,Z 493.686,A -85,B 0,C 180,E1 -523.906,E2 -523.906} C_VEL
LIN {X 0,Y 608.457,Z 493.692,A -85,B 0,C 180,E1 -526.643,E2 -526.643} C_VEL
LIN {X 0,Y 608.469,Z 493.689,A -85,B 0,C 180,E1 -529.35,E2 -529.35} C_VEL
LIN {X 0,Y 608.472,Z 493.685,A -85,B 0,C 180,E1 -532.033,E2 -532.033} C_VEL
LIN {X 0,Y 608.462,Z 493.692,A -85,B 0,C 180,E1 -534.698,E2 -534.698} C_VEL
LIN {X 0,Y 608.485,Z 493.688,A -85,B 0,C 180,E1 -537.352,E2 -537.352} C_VEL
LIN {X 0,Y 608.467,Z 493.685,A -85,B 0,C 180,E1 -540,E2 -540} C_VEL
LIN {X 0,Y 608.481,Z 493.688,A -85,B 0,C 180,E1 -542.648,E2 -542.648} C_VEL
LIN {X 0,Y 608.47,Z 493.691,A -85,B 0,C 180,E1 -545.301,E2 -545.301} C_VEL
LIN {X 0,Y 608.471,Z 493.685,A -85,B 0,C 180,E1 -547.967,E2 -547.967} C_VEL
LIN {X 0,Y 608.459,Z 493.69,A -85,B 0,C 180,E1 -549.472,E2 -549.472} C_VEL
LIN {X 0,Y 607.773,Z 493.774,A -85,B 0,C 180,E1 -550.025,E2 -550.025} C_VEL
LIN {X 0,Y 604.914,Z 494.136,A -85,B 0,C 180,E1 -550.922,E2 -550.922} C_VEL
LIN {X 0,Y 602.514,Z 494.43,A -85,B 0,C 180,E1 -551.643,E2 -551.643} C_VEL
LIN {X 0,Y 601.489,Z 494.555,A -85,B 0,C 180,E1 -552.2,E2 -552.2} C_VEL
LIN {X 0,Y 601.407,Z 494.566,A -85,B 0,C 180,E1 -552.388,E2 -552.388} C_VEL
LIN {X 0,Y 601.43,Z 494.569,A -85,B 0,C 180,E1 -554.897,E2 -554.897} C_VEL
LIN {X 0,Y 601.398,Z 494.568,A -85,B 0,C 180,E1 -557.688,E2 -557.688} C_VEL
LIN {X 0,Y 601.427,Z 494.564,A -85,B 0,C 180,E1 -560.522,E2 -560.522} C_VEL
LIN {X 0,Y 601.418,Z 494.57,A -85,B 0,C 180,E1 -563.41,E2 -563.41} C_VEL
LIN {X 0,Y 601.4,Z 494.566,A -85,B 0,C 180,E1 -566.363,E2 -566.363} C_VEL
LIN {X 0,Y 601.436,Z 494.565,A -85,B 0,C 180,E1 -568.791,E2 -568.791} C_VEL
LIN {X 0,Y 601.436,Z 494.568,A -85,B 0,C 180,E1 -571.459,E2 -571.459} C_VEL
LIN {X 0,Y 601.43,Z 494.563,A -85,B 0,C 180,E1 -574.118,E2 -574.118} C_VEL
LIN {X 0,Y 601.479,Z 494.676,A -85,B 0,C 180,E1 -574.622,E2 -574.622} C_VEL
LIN {X 0,Y 601.439,Z 510.977,A -85,B 0,C 180,E1 -577.629,E2 -577.629} C_VEL
LIN {X 0,Y 601.397,Z 517.839,A -85,B 0,C 180,E1 -578.882,E2 -578.882} C_VEL
LIN {X 0,Y 601.672,Z 522.811,A -85,B 0,C 180,E1 -578.959,E2 -578.959} C_VEL
LIN {X 0,Y 601.611,Z 624.234,A -85,B 0,C 180,E1 -580.19,E2 -580.19} C_VEL
LIN {X 0,Y 601.563,Z 637.786,A -85,B 0,C 180,E1 -580.499,E2 -580.499} C_VEL
LIN {X 0,Y 601.555,Z 650.143,A -85,B 0,C 180,E1 -580.918,E2 -580.918} C_VEL
LIN {X 0,Y 601.52,Z 661.926,A -85,B 0,C 180,E1 -581.457,E2 -581.457} C_VEL
LIN {X 0,Y 601.487,Z 672.835,A -85,B 0,C 180,E1 -582.097,E2 -582.097} C_VEL
LIN {X 0,Y 601.429,Z 683.752,A -85,B 0,C 180,E1 -582.896,E2 -582.896} C_VEL
LIN {X 0,Y 601.416,Z 692.699,A -85,B 0,C 180,E1 -583.702,E2 -583.702} C_VEL
LIN {X 0,Y 601.387,Z 700.314,A -85,B 0,C 180,E1 -584.533,E2 -584.533} C_VEL
LIN {X 0,Y 601.388,Z 707.469,A -85,B 0,C 180,E1 -585.48,E2 -585.48} C_VEL
LIN {X 0,Y 601.344,Z 714.556,A -85,B 0,C 180,E1 -586.657,E2 -586.657} C_VEL
LIN {X 0,Y 601.36,Z 719.93,A -85,B 0,C 180,E1 -587.823,E2 -587.823} C_VEL
LIN {X 0,Y 601.331,Z 723.186,A -85,B 0,C 180,E1 -588.768,E2 -588.768} C_VEL
LIN {X 0,Y 601.32,Z 726.141,A -85,B 0,C 180,E1 -589.999,E2 -589.999} C_VEL
LIN {X 0,Y 601.311,Z 727.372,A -85,B 0,C 180,E1 -590.867,E2 -590.867} C_VEL
LIN {X 0,Y 601.326,Z 727.932,A -85,B 0,C 180,E1 -591.726,E2 -591.726} C_VEL
LIN {X 0,Y 601.327,Z 727.842,A -85,B 0,C 180,E1 -592.631,E2 -592.631} C_VEL
LIN {X 0,Y 601.312,Z 726.701,A -85,B 0,C 180,E1 -593.75,E2 -593.75} C_VEL
LIN {X 0,Y 601.334,Z 723.916,A -85,B 0,C 180,E1 -595.064,E2 -595.064} C_VEL
LIN {X 0,Y 601.337,Z 720.636,A -85,B 0,C 180,E1 -596.077,E2 -596.077} C_VEL
LIN {X 0,Y 601.361,Z 715.303,A -85,B 0,C 180,E1 -597.293,E2 -597.293} C_VEL
LIN {X 0,Y 601.392,Z 709.704,A -85,B 0,C 180,E1 -598.273,E2 -598.273} C_VEL
LIN {X 0,Y 601.406,Z 702.761,A -85,B 0,C 180,E1 -599.253,E2 -599.253} C_VEL
LIN {X 0,Y 601.411,Z 694.296,A -85,B 0,C 180,E1 -600.222,E2 -600.222} C_VEL
LIN {X 0,Y 601.438,Z 684.831,A -85,B 0,C 180,E1 -601.106,E2 -601.106} C_VEL
LIN {X 0,Y 601.461,Z 674.981,A -85,B 0,C 180,E1 -601.851,E2 -601.851} C_VEL
LIN {X 0,Y 601.476,Z 663.395,A -85,B 0,C 180,E1 -602.554,E2 -602.554} C_VEL
LIN {X 0,Y 601.551,Z 651.233,A -85,B 0,C 180,E1 -603.129,E2 -603.129} C_VEL
LIN {X 0,Y 601.55,Z 638.42,A -85,B 0,C 180,E1 -603.574,E2 -603.574} C_VEL
LIN {X 0,Y 601.613,Z 625.199,A -85,B 0,C 180,E1 -603.882,E2 -603.882} C_VEL
LIN {X 0,Y 601.621,Z 590.108,A -85,B 0,C 180,E1 -604.326,E2 -604.326} C_VEL
LIN {X 0,Y 601.486,Z 518.451,A -85,B 0,C 180,E1 -605.188,E2 -605.188} C_VEL
LIN {X 0,Y 601.417,Z 517.851,A -85,B 0,C 180,E1 -605.205,E2 -605.205} C_VEL
LIN {X 0,Y 601.446,Z 502.375,A -85,B 0,C 180,E1 -608.043,E2 -608.043} C_VEL
LIN {X 0,Y 601.422,Z 494.565,A -85,B 0,C 180,E1 -609.523,E2 -609.523} C_VEL
LIN {X 0,Y 601.397,Z 494.569,A -85,B 0,C 180,E1 -612.312,E2 -612.312} C_VEL
LIN {X 0,Y 601.416,Z 494.567,A -85,B 0,C 180,E1 -614.409,E2 -614.409} C_VEL
LIN {X 0,Y 601.417,Z 494.569,A -85,B 0,C 180,E1 -617.172,E2 -617.172} C_VEL
LIN {X 0,Y 601.431,Z 494.562,A -85,B 0,C 180,E1 -619.905,E2 -619.905} C_VEL
LIN {X 0,Y 601.454,Z 494.565,A -85,B 0,C 180,E1 -622.615,E2 -622.615} C_VEL
LIN {X 0,Y 601.416,Z 494.567,A -85,B 0,C 180,E1 -625.308,E2 -625.308} C_VEL
LIN {X 0,Y 601.434,Z 494.561,A -85,B 0,C 180,E1 -627.991,E2 -627.991} C_VEL
LIN {X 0,Y 601.449,Z 494.566,A -85,B 0,C 180,E1 -630.67,E2 -630.67} C_VEL
LIN {X 0,Y 601.427,Z 494.566,A -85,B 0,C 180,E1 -633.349,E2 -633.349} C_VEL
LIN {X 0,Y 601.434,Z 494.561,A -85,B 0,C 180,E1 -636.037,E2 -636.037} C_VEL
LIN {X 0,Y 601.432,Z 494.569,A -85,B 0,C 180,E1 -638.737,E2 -638.737} C_VEL
LIN {X 0,Y 601.434,Z 494.564,A -85,B 0,C 180,E1 -641.458,E2 -641.458} C_VEL
LIN {X 0,Y 601.417,Z 494.564,A -85,B 0,C 180,E1 -644.205,E2 -644.205} C_VEL
LIN {X 0,Y 601.43,Z 494.573,A -85,B 0,C 180,E1 -646.986,E2 -646.986} C_VEL
LIN {X 0,Y 601.406,Z 494.565,A -85,B 0,C 180,E1 -649.809,E2 -649.809} C_VEL
LIN {X 0,Y 601.407,Z 494.57,A -85,B 0,C 180,E1 -652.683,E2 -652.683} C_VEL
LIN {X 0,Y 601.403,Z 494.574,A -85,B 0,C 180,E1 -654.878,E2 -654.878} C_VEL
LIN {X 0,Y 601.42,Z 494.563,A -85,B 0,C 180,E1 -657.867,E2 -657.867} C_VEL
LIN {X 0,Y 601.443,Z 494.56,A -85,B 0,C 180,E1 -660.162,E2 -660.162} C_VEL
LIN {X 0,Y 601.421,Z 494.568,A -85,B 0,C 180,E1 -662.716,E2 -662.716} C_VEL
LIN {X 0,Y 601.405,Z 494.574,A -85,B 0,C 180,E1 -665.114,E2 -665.114} C_VEL
LIN {X 0,Y 601.432,Z 494.566,A -85,B 0,C 180,E1 -667.418,E2 -667.418} C_VEL
LIN {X 0,Y 601.409,Z 494.564,A -85,B 0,C 180,E1 -669.994,E2 -669.994} C_VEL
LIN {X 0,Y 601.433,Z 494.566,A -85,B 0,C 180,E1 -672.667,E2 -672.667} C_VEL
LIN {X 0,Y 601.417,Z 494.567,A -85,B 0,C 180,E1 -675.482,E2 -675.482} C_VEL
LIN {X 0,Y 601.421,Z 494.564,A -85,B 0,C 180,E1 -678.406,E2 -678.406} C_VEL
LIN {X 0,Y 601.436,Z 494.568,A -85,B 0,C 180,E1 -680.876,E2 -680.876} C_VEL
LIN {X 0,Y 601.437,Z 494.562,A -85,B 0,C 180,E1 -683.733,E2 -683.733} C_VEL
LIN {X 0,Y 601.429,Z 494.562,A -85,B 0,C 180,E1 -686.063,E2 -686.063} C_VEL
LIN {X 0,Y 601.434,Z 494.563,A -85,B 0,C 180,E1 -688.541,E2 -688.541} C_VEL
LIN {X 0,Y 601.432,Z 494.568,A -85,B 0,C 180,E1 -691.374,E2 -691.374} C_VEL
LIN {X 0,Y 601.416,Z 494.563,A -85,B 0,C 180,E1 -694.129,E2 -694.129} C_VEL
LIN {X 0,Y 601.419,Z 494.565,A -85,B 0,C 180,E1 -696.59,E2 -696.59} C_VEL
LIN {X 0,Y 601.43,Z 494.567,A -85,B 0,C 180,E1 -699.479,E2 -699.479} C_VEL
LIN {X 0,Y 601.395,Z 494.566,A -85,B 0,C 180,E1 -702.312,E2 -702.312} C_VEL
LIN {X 0,Y 601.411,Z 494.565,A -85,B 0,C 180,E1 -704.409,E2 -704.409} C_VEL
LIN {X 0,Y 601.423,Z 494.574,A -85,B 0,C 180,E1 -707.172,E2 -707.172} C_VEL
LIN {X 0,Y 601.429,Z 494.563,A -85,B 0,C 180,E1 -709.905,E2 -709.905} C_VEL
LIN {X 0,Y 601.447,Z 494.562,A -85,B 0,C 180,E1 -712.615,E2 -712.615} C_VEL
LIN {X 0,Y 601.432,Z 494.57,A -85,B 0,C 180,E1 -715.308,E2 -715.308} C_VEL
LIN {X 0,Y 601.416,Z 494.564,A -85,B 0,C 180,E1 -717.991,E2 -717.991} C_VEL
LIN {X 0,Y 601.45,Z 494.562,A -85,B 0,C 180,E1 -720.67,E2 -720.67} C_VEL
LIN {X 0,Y 601.436,Z 494.57,A -85,B 0,C 180,E1 -723.35,E2 -723.35} C_VEL
LIN {X 0,Y 601.426,Z 494.563,A -85,B 0,C 180,E1 -726.037,E2 -726.037} C_VEL
LIN {X 0,Y 601.439,Z 494.563,A -85,B 0,C 180,E1 -728.738,E2 -728.738} C_VEL
LIN {X 0,Y 601.431,Z 494.569,A -85,B 0,C 180,E1 -731.459,E2 -731.459} C_VEL
LIN {X 0,Y 601.41,Z 494.564,A -85,B 0,C 180,E1 -734.206,E2 -734.206} C_VEL
LIN {X 0,Y 601.432,Z 494.568,A -85,B 0,C 180,E1 -736.986,E2 -736.986} C_VEL
LIN {X 0,Y 601.405,Z 494.567,A -85,B 0,C 180,E1 -739.81,E2 -739.81} C_VEL
LIN {X 0,Y 601.406,Z 494.567,A -85,B 0,C 180,E1 -742.684,E2 -742.684} C_VEL
LIN {X 0,Y 601.401,Z 494.569,A -85,B 0,C 180,E1 -744.879,E2 -744.879} C_VEL
LIN {X 0,Y 601.418,Z 494.565,A -85,B 0,C 180,E1 -747.868,E2 -747.868} C_VEL
LIN {X 0,Y 601.441,Z 494.561,A -85,B 0,C 180,E1 -750.164,E2 -750.164} C_VEL
LIN {X 0,Y 601.42,Z 494.565,A -85,B 0,C 180,E1 -752.717,E2 -752.717} C_VEL
LIN {X 0,Y 601.418,Z 494.571,A -85,B 0,C 180,E1 -755.117,E2 -755.117} C_VEL
LIN {X 0,Y 601.432,Z 494.571,A -85,B 0,C 180,E1 -757.42,E2 -757.42} C_VEL
LIN {X 0,Y 601.408,Z 494.566,A -85,B 0,C 180,E1 -759.996,E2 -759.996} C_VEL
LIN {X 0,Y 601.409,Z 494.566,A -85,B 0,C 180,E1 -762.671,E2 -762.671} C_VEL
LIN {X 0,Y 601.422,Z 494.571,A -85,B 0,C 180,E1 -765.483,E2 -765.483} C_VEL
LIN {X 0,Y 601.424,Z 494.562,A -85,B 0,C 180,E1 -768.407,E2 -768.407} C_VEL
LIN {X 0,Y 601.436,Z 494.564,A -85,B 0,C 180,E1 -770.877,E2 -770.877} C_VEL
LIN {X 0,Y 601.431,Z 494.566,A -85,B 0,C 180,E1 -773.736,E2 -773.736} C_VEL
LIN {X 0,Y 601.427,Z 494.563,A -85,B 0,C 180,E1 -776.687,E2 -776.687} C_VEL
LIN {X 0,Y 601.434,Z 494.567,A -85,B 0,C 180,E1 -779.06,E2 -779.06} C_VEL
LIN {X 0,Y 601.432,Z 494.573,A -85,B 0,C 180,E1 -781.374,E2 -781.374} C_VEL
LIN {X 0,Y 601.402,Z 494.573,A -85,B 0,C 180,E1 -783.637,E2 -783.637} C_VEL
LIN {X 0,Y 601.425,Z 494.583,A -85,B 0,C 180,E1 -786.362,E2 -786.362} C_VEL
LIN {X 0,Y 601.748,Z 497.654,A -85,B 0,C 180,E1 -786.786,E2 -786.786} C_VEL
LIN {X 0,Y 601.642,Z 519.489,A -85,B 0,C 180,E1 -789.665,E2 -789.665} C_VEL
LIN {X 0,Y 601.547,Z 541.325,A -85,B 0,C 180,E1 -792.492,E2 -792.492} C_VEL
LIN {X 0,Y 601.473,Z 563.16,A -85,B 0,C 180,E1 -795.278,E2 -795.278} C_VEL
LIN {X 0,Y 601.471,Z 575.357,A -85,B 0,C 180,E1 -796.819,E2 -796.819} C_VEL
LIN {X 0,Y 601.659,Z 602.999,A -85,B 0,C 180,E1 -797.156,E2 -797.156} C_VEL
LIN {X 0,Y 601.603,Z 683.962,A -85,B 0,C 180,E1 -798.14,E2 -798.14} C_VEL
LIN {X 0,Y 601.572,Z 697.227,A -85,B 0,C 180,E1 -798.438,E2 -798.438} C_VEL
LIN {X 0,Y 601.547,Z 708.928,A -85,B 0,C 180,E1 -798.826,E2 -798.826} C_VEL
LIN {X 0,Y 601.515,Z 719.928,A -85,B 0,C 180,E1 -799.311,E2 -799.311} C_VEL
LIN {X 0,Y 601.466,Z 730.584,A -85,B 0,C 180,E1 -799.906,E2 -799.906} C_VEL
LIN {X 0,Y 601.445,Z 741.478,A -85,B 0,C 180,E1 -800.67,E2 -800.67} C_VEL
LIN {X 0,Y 601.429,Z 752.114,A -85,B 0,C 180,E1 -801.601,E2 -801.601} C_VEL
LIN {X 0,Y 601.418,Z 759.962,A -85,B 0,C 180,E1 -802.446,E2 -802.446} C_VEL
LIN {X 0,Y 601.37,Z 767.226,A -85,B 0,C 180,E1 -803.398,E2 -803.398} C_VEL
LIN {X 0,Y 601.371,Z 772.867,A -85,B 0,C 180,E1 -804.299,E2 -804.299} C_VEL
LIN {X 0,Y 601.337,Z 777.951,A -85,B 0,C 180,E1 -805.307,E2 -805.307} C_VEL
LIN {X 0,Y 601.367,Z 781.896,A -85,B 0,C 180,E1 -806.315,E2 -806.315} C_VEL
LIN {X 0,Y 601.325,Z 784.809,A -85,B 0,C 180,E1 -807.321,E2 -807.321} C_VEL
LIN {X 0,Y 601.34,Z 786.202,A -85,B 0,C 180,E1 -807.991,E2 -807.991} C_VEL
LIN {X 0,Y 601.339,Z 787.784,A -85,B 0,C 180,E1 -809.33,E2 -809.33} C_VEL
LIN {X 0,Y 601.335,Z 788,A -85,B 0,C 180,E1 -810,E2 -810} C_VEL
LIN {X 0,Y 601.348,Z 787.184,A -85,B 0,C 180,E1 -811.339,E2 -811.339} C_VEL
LIN {X 0,Y 601.34,Z 786.202,A -85,B 0,C 180,E1 -812.009,E2 -812.009} C_VEL
LIN {X 0,Y 601.325,Z 784.809,A -85,B 0,C 180,E1 -812.679,E2 -812.679} C_VEL
LIN {X 0,Y 601.367,Z 781.896,A -85,B 0,C 180,E1 -813.685,E2 -813.685} C_VEL
LIN {X 0,Y 601.337,Z 777.95,A -85,B 0,C 180,E1 -814.693,E2 -814.693} C_VEL
LIN {X 0,Y 601.372,Z 771.878,A -85,B 0,C 180,E1 -815.869,E2 -815.869} C_VEL
LIN {X 0,Y 601.382,Z 765.237,A -85,B 0,C 180,E1 -816.88,E2 -816.88} C_VEL
LIN {X 0,Y 601.4,Z 756.991,A -85,B 0,C 180,E1 -817.892,E2 -817.892} C_VEL
LIN {X 0,Y 601.436,Z 748.539,A -85,B 0,C 180,E1 -818.737,E2 -818.737} C_VEL
LIN {X 0,Y 601.442,Z 738.095,A -85,B 0,C 180,E1 -819.585,E2 -819.585} C_VEL
LIN {X 0,Y 601.484,Z 727.761,A -85,B 0,C 180,E1 -820.264,E2 -820.264} C_VEL
LIN {X 0,Y 601.537,Z 716.902,A -85,B 0,C 180,E1 -820.836,E2 -820.836} C_VEL
LIN {X 0,Y 601.559,Z 704.382,A -85,B 0,C 180,E1 -821.34,E2 -821.34} C_VEL
LIN {X 0,Y 601.566,Z 691.364,A -85,B 0,C 180,E1 -821.712,E2 -821.712} C_VEL
LIN {X 0,Y 601.61,Z 678.106,A -85,B 0,C 180,E1 -821.946,E2 -821.946} C_VEL
LIN {X 0,Y 601.565,Z 576.169,A -85,B 0,C 180,E1 -823.168,E2 -823.168} C_VEL
LIN {X 0,Y 601.477,Z 575.272,A -85,B 0,C 180,E1 -823.192,E2 -823.192} C_VEL
LIN {X 0,Y 601.525,Z 552.242,A -85,B 0,C 180,E1 -826.11,E2 -826.11} C_VEL
LIN {X 0,Y 601.605,Z 529.042,A -85,B 0,C 180,E1 -829.092,E2 -829.092} C_VEL
LIN {X 0,Y 601.673,Z 507.207,A -85,B 0,C 180,E1 -831.949,E2 -831.949} C_VEL
LIN {X 0,Y 601.742,Z 496.289,A -85,B 0,C 180,E1 -833.396,E2 -833.396} C_VEL
LIN {X 0,Y 601.422,Z 494.567,A -85,B 0,C 180,E1 -833.661,E2 -833.661} C_VEL
LIN {X 0,Y 601.402,Z 494.573,A -85,B 0,C 180,E1 -836.363,E2 -836.363} C_VEL
LIN {X 0,Y 601.438,Z 494.569,A -85,B 0,C 180,E1 -838.788,E2 -838.788} C_VEL
LIN {X 0,Y 601.413,Z 494.564,A -85,B 0,C 180,E1 -841.725,E2 -841.725} C_VEL
LIN {X 0,Y 601.43,Z 494.565,A -85,B 0,C 180,E1 -844.117,E2 -844.117} C_VEL
LIN {X 0,Y 601.416,Z 494.573,A -85,B 0,C 180,E1 -846.581,E2 -846.581} C_VEL
LIN {X 0,Y 601.437,Z 494.561,A -85,B 0,C 180,E1 -849.535,E2 -849.535} C_VEL
LIN {X 0,Y 601.436,Z 494.57,A -85,B 0,C 180,E1 -852.593,E2 -852.593} C_VEL
LIN {X 0,Y 601.422,Z 494.563,A -85,B 0,C 180,E1 -855.481,E2 -855.481} C_VEL
LIN {X 0,Y 601.421,Z 494.568,A -85,B 0,C 180,E1 -858.406,E2 -858.406} C_VEL
LIN {X 0,Y 601.437,Z 494.57,A -85,B 0,C 180,E1 -860.875,E2 -860.875} C_VEL
LIN {X 0,Y 601.44,Z 494.56,A -85,B 0,C 180,E1 -863.733,E2 -863.733} C_VEL
LIN {X 0,Y 601.43,Z 494.562,A -85,B 0,C 180,E1 -866.063,E2 -866.063} C_VEL
LIN {X 0,Y 601.437,Z 494.567,A -85,B 0,C 180,E1 -868.54,E2 -868.54} C_VEL
LIN {X 0,Y 601.432,Z 494.564,A -85,B 0,C 180,E1 -871.373,E2 -871.373} C_VEL
LIN {X 0,Y 601.405,Z 494.565,A -85,B 0,C 180,E1 -873.636,E2 -873.636} C_VEL
LIN {X 0,Y 601.419,Z 494.569,A -85,B 0,C 180,E1 -876.589,E2 -876.589} C_VEL
LIN {X 0,Y 601.429,Z 494.564,A -85,B 0,C 180,E1 -879.478,E2 -879.478} C_VEL
LIN {X 0,Y 601.392,Z 494.568,A -85,B 0,C 180,E1 -882.311,E2 -882.311} C_VEL
LIN {X 0,Y 601.414,Z 494.566,A -85,B 0,C 180,E1 -884.408,E2 -884.408} C_VEL
LIN {X 0,Y 601.421,Z 494.57,A -85,B 0,C 180,E1 -887.172,E2 -887.172} C_VEL
LIN {X 0,Y 601.429,Z 494.562,A -85,B 0,C 180,E1 -889.905,E2 -889.905} C_VEL
LIN {X 0,Y 601.448,Z 494.564,A -85,B 0,C 180,E1 -892.615,E2 -892.615} C_VEL
LIN {X 0,Y 601.431,Z 494.567,A -85,B 0,C 180,E1 -895.308,E2 -895.308} C_VEL
LIN {X 0,Y 601.416,Z 494.563,A -85,B 0,C 180,E1 -897.991,E2 -897.991} C_VEL
LIN {X 0,Y 601.449,Z 494.564,A -85,B 0,C 180,E1 -900.669,E2 -900.669} C_VEL
LIN {X 0,Y 601.435,Z 494.566,A -85,B 0,C 180,E1 -903.349,E2 -903.349} C_VEL
LIN {X 0,Y 601.426,Z 494.562,A -85,B 0,C 180,E1 -906.037,E2 -906.037} C_VEL
LIN {X 0,Y 601.437,Z 494.566,A -85,B 0,C 180,E1 -908.737,E2 -908.737} C_VEL
LIN {X 0,Y 601.431,Z 494.566,A -85,B 0,C 180,E1 -911.458,E2 -911.458} C_VEL
LIN {X 0,Y 601.407,Z 494.566,A -85,B 0,C 180,E1 -912.388,E2 -912.388} C_VEL
LIN {X 0,Y 600.747,Z 494.655,A -85,B 0,C 180,E1 -912.948,E2 -912.948} C_VEL
LIN {X 0,Y 597.898,Z 495.014,A -85,B 0,C 180,E1 -913.855,E2 -913.855} C_VEL
LIN {X 0,Y 595.485,Z 495.315,A -85,B 0,C 180,E1 -914.586,E2 -914.586} C_VEL
LIN {X 0,Y 594.446,Z 495.442,A -85,B 0,C 180,E1 -915.149,E2 -915.149} C_VEL
LIN {X 0,Y 594.36,Z 495.448,A -85,B 0,C 180,E1 -915.34,E2 -915.34} C_VEL
LIN {X 0,Y 594.377,Z 495.441,A -85,B 0,C 180,E1 -917.904,E2 -917.904} C_VEL
LIN {X 0,Y 594.376,Z 495.447,A -85,B 0,C 180,E1 -920.919,E2 -920.919} C_VEL
LIN {X 0,Y 594.385,Z 495.442,A -85,B 0,C 180,E1 -923.704,E2 -923.704} C_VEL
LIN {X 0,Y 594.381,Z 495.444,A -85,B 0,C 180,E1 -926.699,E2 -926.699} C_VEL
LIN {X 0,Y 594.379,Z 495.448,A -85,B 0,C 180,E1 -928.998,E2 -928.998} C_VEL
LIN {X 0,Y 594.386,Z 495.444,A -85,B 0,C 180,E1 -931.646,E2 -931.646} C_VEL
LIN {X 0,Y 594.401,Z 495.583,A -85,B 0,C 180,E1 -934.578,E2 -934.578} C_VEL
LIN {X 0,Y 594.408,Z 508.982,A -85,B 0,C 180,E1 -937.085,E2 -937.085} C_VEL
LIN {X 0,Y 594.359,Z 517.857,A -85,B 0,C 180,E1 -938.727,E2 -938.727} C_VEL
LIN {X 0,Y 594.756,Z 522.71,A -85,B 0,C 180,E1 -938.803,E2 -938.803} C_VEL
LIN {X 0,Y 594.663,Z 624.134,A -85,B 0,C 180,E1 -940.047,E2 -940.047} C_VEL
LIN {X 0,Y 594.602,Z 637.453,A -85,B 0,C 180,E1 -940.352,E2 -940.352} C_VEL
LIN {X 0,Y 594.585,Z 649.886,A -85,B 0,C 180,E1 -940.776,E2 -940.776} C_VEL
LIN {X 0,Y 594.535,Z 660.998,A -85,B 0,C 180,E1 -941.282,E2 -941.282} C_VEL
LIN {X 0,Y 594.463,Z 672.077,A -85,B 0,C 180,E1 -941.927,E2 -941.927} C_VEL
LIN {X 0,Y 594.384,Z 683.561,A -85,B 0,C 180,E1 -942.771,E2 -942.771} C_VEL
LIN {X 0,Y 594.386,Z 693.67,A -85,B 0,C 180,E1 -943.704,E2 -943.704} C_VEL
LIN {X 0,Y 594.323,Z 702.083,A -85,B 0,C 180,E1 -944.665,E2 -944.665} C_VEL
LIN {X 0,Y 594.306,Z 709.805,A -85,B 0,C 180,E1 -945.758,E2 -945.758} C_VEL
LIN {X 0,Y 594.275,Z 716.334,A -85,B 0,C 180,E1 -946.95,E2 -946.95} C_VEL
LIN {X 0,Y 594.269,Z 721.358,A -85,B 0,C 180,E1 -948.163,E2 -948.163} C_VEL
LIN {X 0,Y 594.247,Z 725.015,A -85,B 0,C 180,E1 -949.424,E2 -949.424} C_VEL
LIN {X 0,Y 594.213,Z 726.683,A -85,B 0,C 180,E1 -950.308,E2 -950.308} C_VEL
LIN {X 0,Y 594.203,Z 727.749,A -85,B 0,C 180,E1 -951.317,E2 -951.317} C_VEL
LIN {X 0,Y 594.222,Z 727.922,A -85,B 0,C 180,E1 -952.412,E2 -952.412} C_VEL
LIN {X 0,Y 594.229,Z 726.738,A -85,B 0,C 180,E1 -953.748,E2 -953.748} C_VEL
LIN {X 0,Y 594.223,Z 724.955,A -85,B 0,C 180,E1 -954.693,E2 -954.693} C_VEL
LIN {X 0,Y 594.261,Z 721.536,A -85,B 0,C 180,E1 -955.878,E2 -955.878} C_VEL
LIN {X 0,Y 594.259,Z 716.499,A -85,B 0,C 180,E1 -957.106,E2 -957.106} C_VEL
LIN {X 0,Y 594.296,Z 710.979,A -85,B 0,C 180,E1 -958.136,E2 -958.136} C_VEL
LIN {X 0,Y 594.324,Z 703.532,A -85,B 0,C 180,E1 -959.241,E2 -959.241} C_VEL
LIN {X 0,Y 594.343,Z 695.223,A -85,B 0,C 180,E1 -960.223,E2 -960.223} C_VEL
LIN {X 0,Y 594.384,Z 686.796,A -85,B 0,C 180,E1 -961.041,E2 -961.041} C_VEL
LIN {X 0,Y 594.449,Z 676.356,A -85,B 0,C 180,E1 -961.872,E2 -961.872} C_VEL
LIN {X 0,Y 594.496,Z 665.821,A -85,B 0,C 180,E1 -962.546,E2 -962.546} C_VEL
LIN {X 0,Y 594.545,Z 653.408,A -85,B 0,C 180,E1 -963.167,E2 -963.167} C_VEL
LIN {X 0,Y 594.593,Z 641.407,A -85,B 0,C 180,E1 -963.619,E2 -963.619} C_VEL
LIN {X 0,Y 594.648,Z 628.313,A -85,B 0,C 180,E1 -963.964,E2 -963.964} C_VEL
LIN {X 0,Y 594.674,Z 611.554,A -85,B 0,C 180,E1 -964.212,E2 -964.212} C_VEL
LIN {X 0,Y 594.617,Z 519.443,A -85,B 0,C 180,E1 -965.33,E2 -965.33} C_VEL
LIN {X 0,Y 594.357,Z 517.885,A -85,B 0,C 180,E1 -965.358,E2 -965.358} C_VEL
LIN {X 0,Y 594.414,Z 502.924,A -85,B 0,C 180,E1 -968.135,E2 -968.135} C_VEL
LIN {X 0,Y 594.386,Z 495.443,A -85,B 0,C 180,E1 -969.541,E2 -969.541} C_VEL
LIN {X 0,Y 594.377,Z 495.442,A -85,B 0,C 180,E1 -972.096,E2 -972.096} C_VEL
LIN {X 0,Y 594.368,Z 495.443,A -85,B 0,C 180,E1 -974.219,E2 -974.219} C_VEL
LIN {X 0,Y 594.366,Z 495.45,A -85,B 0,C 180,E1 -977.017,E2 -977.017} C_VEL
LIN {X 0,Y 594.39,Z 495.439,A -85,B 0,C 180,E1 -979.784,E2 -979.784} C_VEL
LIN {X 0,Y 594.402,Z 495.442,A -85,B 0,C 180,E1 -982.527,E2 -982.527} C_VEL
LIN {X 0,Y 594.387,Z 495.444,A -85,B 0,C 180,E1 -985.252,E2 -985.252} C_VEL
LIN {X 0,Y 594.403,Z 495.437,A -85,B 0,C 180,E1 -987.967,E2 -987.967} C_VEL
LIN {X 0,Y 594.42,Z 495.441,A -85,B 0,C 180,E1 -990.677,E2 -990.677} C_VEL
LIN {X 0,Y 594.379,Z 495.443,A -85,B 0,C 180,E1 -993.389,E2 -993.389} C_VEL
LIN {X 0,Y 594.388,Z 495.439,A -85,B 0,C 180,E1 -996.109,E2 -996.109} C_VEL
LIN {X 0,Y 594.394,Z 495.447,A -85,B 0,C 180,E1 -998.842,E2 -998.842} C_VEL
LIN {X 0,Y 594.393,Z 495.44,A -85,B 0,C 180,E1 -1001.595,E2 -1001.595} C_VEL
LIN {X 0,Y 594.387,Z 495.441,A -85,B 0,C 180,E1 -1004.377,E2 -1004.377} C_VEL
LIN {X 0,Y 594.388,Z 495.446,A -85,B 0,C 180,E1 -1007.193,E2 -1007.193} C_VEL
LIN {X 0,Y 594.375,Z 495.441,A -85,B 0,C 180,E1 -1010.053,E2 -1010.053} C_VEL
LIN {X 0,Y 594.36,Z 495.453,A -85,B 0,C 180,E1 -1012.967,E2 -1012.967} C_VEL
LIN {X 0,Y 594.373,Z 495.448,A -85,B 0,C 180,E1 -1015.193,E2 -1015.193} C_VEL
LIN {X 0,Y 594.38,Z 495.443,A -85,B 0,C 180,E1 -1017.526,E2 -1017.526} C_VEL
LIN {X 0,Y 594.396,Z 495.439,A -85,B 0,C 180,E1 -1020.33,E2 -1020.33} C_VEL
LIN {X 0,Y 594.374,Z 495.451,A -85,B 0,C 180,E1 -1022.95,E2 -1022.95} C_VEL
LIN {X 0,Y 594.375,Z 495.445,A -85,B 0,C 180,E1 -1025.406,E2 -1025.406} C_VEL
LIN {X 0,Y 594.385,Z 495.439,A -85,B 0,C 180,E1 -1027.94,E2 -1027.94} C_VEL
LIN {X 0,Y 594.387,Z 495.446,A -85,B 0,C 180,E1 -1030.824,E2 -1030.824} C_VEL
LIN {X 0,Y 594.38,Z 495.447,A -85,B 0,C 180,E1 -1033.297,E2 -1033.297} C_VEL
LIN {X 0,Y 594.373,Z 495.441,A -85,B 0,C 180,E1 -1036.159,E2 -1036.159} C_VEL
LIN {X 0,Y 594.376,Z 495.45,A -85,B 0,C 180,E1 -1039.177,E2 -1039.177} C_VEL
LIN {X 0,Y 594.381,Z 495.44,A -85,B 0,C 180,E1 -1042.059,E2 -1042.059} C_VEL
LIN {X 0,Y 594.382,Z 495.444,A -85,B 0,C 180,E1 -1044.67,E2 -1044.67} C_VEL
LIN {X 0,Y 594.371,Z 495.452,A -85,B 0,C 180,E1 -1047.088,E2 -1047.088} C_VEL
LIN {X 0,Y 594.391,Z 495.441,A -85,B 0,C 180,E1 -1049.669,E2 -1049.669} C_VEL
LIN {X 0,Y 594.38,Z 495.442,A -85,B 0,C 180,E1 -1052.54,E2 -1052.54} C_VEL
LIN {X 0,Y 594.376,Z 495.446,A -85,B 0,C 180,E1 -1054.807,E2 -1054.807} C_VEL
LIN {X 0,Y 594.358,Z 495.451,A -85,B 0,C 180,E1 -1057.263,E2 -1057.263} C_VEL
LIN {X 0,Y 594.372,Z 495.441,A -85,B 0,C 180,E1 -1059.947,E2 -1059.947} C_VEL
LIN {X 0,Y 594.385,Z 495.444,A -85,B 0,C 180,E1 -1062.807,E2 -1062.807} C_VEL
LIN {X 0,Y 594.378,Z 495.442,A -85,B 0,C 180,E1 -1065.826,E2 -1065.826} C_VEL
LIN {X 0,Y 594.386,Z 495.44,A -85,B 0,C 180,E1 -1068.404,E2 -1068.404} C_VEL
LIN {X 0,Y 594.398,Z 495.449,A -85,B 0,C 180,E1 -1071.158,E2 -1071.158} C_VEL
LIN {X 0,Y 594.38,Z 495.441,A -85,B 0,C 180,E1 -1073.892,E2 -1073.892} C_VEL
LIN {X 0,Y 594.382,Z 495.442,A -85,B 0,C 180,E1 -1076.611,E2 -1076.611} C_VEL
LIN {X 0,Y 594.427,Z 495.443,A -85,B 0,C 180,E1 -1079.323,E2 -1079.323} C_VEL
LIN {X 0,Y 594.388,Z 495.439,A -85,B 0,C 180,E1 -1082.033,E2 -1082.033} C_VEL
LIN {X 0,Y 594.401,Z 495.441,A -85,B 0,C 180,E1 -1084.748,E2 -1084.748} C_VEL
LIN {X 0,Y 594.413,Z 495.442,A -85,B 0,C 180,E1 -1087.473,E2 -1087.473} C_VEL
LIN {X 0,Y 594.388,Z 495.439,A -85,B 0,C 180,E1 -1090.216,E2 -1090.216} C_VEL
LIN {X 0,Y 594.372,Z 495.447,A -85,B 0,C 180,E1 -1092.983,E2 -1092.983} C_VEL
LIN {X 0,Y 594.366,Z 495.444,A -85,B 0,C 180,E1 -1095.781,E2 -1095.781} C_VEL
LIN {X 0,Y 594.384,Z 495.441,A -85,B 0,C 180,E1 -1098.618,E2 -1098.618} C_VEL
LIN {X 0,Y 594.366,Z 495.449,A -85,B 0,C 180,E1 -1101.504,E2 -1101.504} C_VEL
LIN {X 0,Y 594.38,Z 495.44,A -85,B 0,C 180,E1 -1104.447,E2 -1104.447} C_VEL
LIN {X 0,Y 594.384,Z 495.441,A -85,B 0,C 180,E1 -1106.7,E2 -1106.7} C_VEL
LIN {X 0,Y 594.379,Z 495.446,A -85,B 0,C 180,E1 -1108.999,E2 -1108.999} C_VEL
LIN {X 0,Y 594.387,Z 495.444,A -85,B 0,C 180,E1 -1111.646,E2 -1111.646} C_VEL
LIN {X 0,Y 594.395,Z 495.439,A -85,B 0,C 180,E1 -1114.579,E2 -1114.579} C_VEL
LIN {X 0,Y 594.383,Z 495.446,A -85,B 0,C 180,E1 -1117.087,E2 -1117.087} C_VEL
LIN {X 0,Y 594.374,Z 495.444,A -85,B 0,C 180,E1 -1119.776,E2 -1119.776} C_VEL
LIN {X 0,Y 594.365,Z 495.442,A -85,B 0,C 180,E1 -1122.376,E2 -1122.376} C_VEL
LIN {X 0,Y 594.36,Z 495.451,A -85,B 0,C 180,E1 -1125.192,E2 -1125.192} C_VEL
LIN {X 0,Y 594.385,Z 495.445,A -85,B 0,C 180,E1 -1127.627,E2 -1127.627} C_VEL
LIN {X 0,Y 594.389,Z 495.439,A -85,B 0,C 180,E1 -1130.322,E2 -1130.322} C_VEL
LIN {X 0,Y 594.385,Z 495.443,A -85,B 0,C 180,E1 -1132.914,E2 -1132.914} C_VEL
LIN {X 0,Y 594.383,Z 495.443,A -85,B 0,C 180,E1 -1135.862,E2 -1135.862} C_VEL
LIN {X 0,Y 594.391,Z 495.44,A -85,B 0,C 180,E1 -1138.652,E2 -1138.652} C_VEL
LIN {X 0,Y 594.383,Z 495.445,A -85,B 0,C 180,E1 -1141.043,E2 -1141.043} C_VEL
LIN {X 0,Y 594.382,Z 495.443,A -85,B 0,C 180,E1 -1143.979,E2 -1143.979} C_VEL
LIN {X 0,Y 594.432,Z 495.607,A -85,B 0,C 180,E1 -1146.206,E2 -1146.206} C_VEL
LIN {X 0,Y 594.87,Z 499.018,A -85,B 0,C 180,E1 -1146.686,E2 -1146.686} C_VEL
LIN {X 0,Y 594.72,Z 520.854,A -85,B 0,C 180,E1 -1149.598,E2 -1149.598} C_VEL
LIN {X 0,Y 594.583,Z 542.689,A -85,B 0,C 180,E1 -1152.458,E2 -1152.458} C_VEL
LIN {X 0,Y 594.476,Z 564.525,A -85,B 0,C 180,E1 -1155.276,E2 -1155.276} C_VEL
LIN {X 0,Y 594.463,Z 575.357,A -85,B 0,C 180,E1 -1156.661,E2 -1156.661} C_VEL
LIN {X 0,Y 594.765,Z 581.535,A -85,B 0,C 180,E1 -1156.744,E2 -1156.744} C_VEL
LIN {X 0,Y 594.654,Z 683.962,A -85,B 0,C 180,E1 -1157.999,E2 -1157.999} C_VEL
LIN {X 0,Y 594.615,Z 697.228,A -85,B 0,C 180,E1 -1158.301,E2 -1158.301} C_VEL
LIN {X 0,Y 594.591,Z 710.378,A -85,B 0,C 180,E1 -1158.75,E2 -1158.75} C_VEL
LIN {X 0,Y 594.538,Z 721.638,A -85,B 0,C 180,E1 -1159.27,E2 -1159.27} C_VEL
LIN {X 0,Y 594.468,Z 733.203,A -85,B 0,C 180,E1 -1159.958,E2 -1159.958} C_VEL
LIN {X 0,Y 594.413,Z 743.599,A -85,B 0,C 180,E1 -1160.73,E2 -1160.73} C_VEL
LIN {X 0,Y 594.383,Z 752.114,A -85,B 0,C 180,E1 -1161.501,E2 -1161.501} C_VEL
LIN {X 0,Y 594.347,Z 759.962,A -85,B 0,C 180,E1 -1162.356,E2 -1162.356} C_VEL
LIN {X 0,Y 594.282,Z 767.814,A -85,B 0,C 180,E1 -1163.409,E2 -1163.409} C_VEL
LIN {X 0,Y 594.289,Z 774.681,A -85,B 0,C 180,E1 -1164.571,E2 -1164.571} C_VEL
LIN {X 0,Y 594.27,Z 779.372,A -85,B 0,C 180,E1 -1165.591,E2 -1165.591} C_VEL
LIN {X 0,Y 594.268,Z 782.956,A -85,B 0,C 180,E1 -1166.61,E2 -1166.61} C_VEL
LIN {X 0,Y 594.226,Z 784.809,A -85,B 0,C 180,E1 -1167.288,E2 -1167.288} C_VEL
LIN {X 0,Y 594.239,Z 786.202,A -85,B 0,C 180,E1 -1167.967,E2 -1167.967} C_VEL
LIN {X 0,Y 594.239,Z 787.784,A -85,B 0,C 180,E1 -1169.322,E2 -1169.322} C_VEL
LIN {X 0,Y 594.236,Z 788,A -85,B 0,C 180,E1 -1170,E2 -1170} C_VEL
LIN {X 0,Y 594.247,Z 787.185,A -85,B 0,C 180,E1 -1171.355,E2 -1171.355} C_VEL
LIN {X 0,Y 594.239,Z 786.202,A -85,B 0,C 180,E1 -1172.033,E2 -1172.033} C_VEL
LIN {X 0,Y 594.226,Z 784.81,A -85,B 0,C 180,E1 -1172.712,E2 -1172.712} C_VEL
LIN {X 0,Y 594.288,Z 781.896,A -85,B 0,C 180,E1 -1173.729,E2 -1173.729} C_VEL
LIN {X 0,Y 594.242,Z 777.95,A -85,B 0,C 180,E1 -1174.749,E2 -1174.749} C_VEL
LIN {X 0,Y 594.304,Z 771.878,A -85,B 0,C 180,E1 -1175.939,E2 -1175.939} C_VEL
LIN {X 0,Y 594.308,Z 765.237,A -85,B 0,C 180,E1 -1176.962,E2 -1176.962} C_VEL
LIN {X 0,Y 594.359,Z 756.991,A -85,B 0,C 180,E1 -1177.986,E2 -1177.986} C_VEL
LIN {X 0,Y 594.382,Z 748.539,A -85,B 0,C 180,E1 -1178.842,E2 -1178.842} C_VEL
LIN {X 0,Y 594.423,Z 738.096,A -85,B 0,C 180,E1 -1179.699,E2 -1179.699} C_VEL
LIN {X 0,Y 594.485,Z 727.763,A -85,B 0,C 180,E1 -1180.386,E2 -1180.386} C_VEL
LIN {X 0,Y 594.56,Z 716.698,A -85,B 0,C 180,E1 -1180.974,E2 -1180.974} C_VEL
LIN {X 0,Y 594.594,Z 704.71,A -85,B 0,C 180,E1 -1181.464,E2 -1181.464} C_VEL
LIN {X 0,Y 594.635,Z 691.363,A -85,B 0,C 180,E1 -1181.85,E2 -1181.85} C_VEL
LIN {X 0,Y 594.688,Z 678.106,A -85,B 0,C 180,E1 -1182.087,E2 -1182.087} C_VEL
LIN {X 0,Y 594.658,Z 576.839,A -85,B 0,C 180,E1 -1183.316,E2 -1183.316} C_VEL
LIN {X 0,Y 594.47,Z 575.272,A -85,B 0,C 180,E1 -1183.35,E2 -1183.35} C_VEL
LIN {X 0,Y 594.551,Z 552.242,A -85,B 0,C 180,E1 -1186.304,E2 -1186.304} C_VEL
LIN {X 0,Y 594.681,Z 529.042,A -85,B 0,C 180,E1 -1189.323,E2 -1189.323} C_VEL
LIN {X 0,Y 594.822,Z 506.061,A -85,B 0,C 180,E1 -1192.368,E2 -1192.368} C_VEL
LIN {X 0,Y 594.818,Z 497.654,A -85,B 0,C 180,E1 -1193.501,E2 -1193.501} C_VEL
LIN {X 0,Y 594.415,Z 495.443,A -85,B 0,C 180,E1 -1193.841,E2 -1193.841} C_VEL
LIN {X 0,Y 594.387,Z 495.449,A -85,B 0,C 180,E1 -1196.699,E2 -1196.699} C_VEL
LIN {X 0,Y 594.381,Z 495.445,A -85,B 0,C 180,E1 -1198.998,E2 -1198.998} C_VEL
LIN {X 0,Y 594.391,Z 495.439,A -85,B 0,C 180,E1 -1201.644,E2 -1201.644} C_VEL
LIN {X 0,Y 594.396,Z 495.448,A -85,B 0,C 180,E1 -1204.578,E2 -1204.578} C_VEL
LIN {X 0,Y 594.387,Z 495.443,A -85,B 0,C 180,E1 -1207.086,E2 -1207.086} C_VEL
LIN {X 0,Y 594.373,Z 495.441,A -85,B 0,C 180,E1 -1209.774,E2 -1209.774} C_VEL
LIN {X 0,Y 594.385,Z 495.445,A -85,B 0,C 180,E1 -1212.373,E2 -1212.373} C_VEL
LIN {X 0,Y 594.359,Z 495.446,A -85,B 0,C 180,E1 -1215.19,E2 -1215.19} C_VEL
LIN {X 0,Y 594.365,Z 495.442,A -85,B 0,C 180,E1 -1217.624,E2 -1217.624} C_VEL
LIN {X 0,Y 594.392,Z 495.442,A -85,B 0,C 180,E1 -1220.32,E2 -1220.32} C_VEL
LIN {X 0,Y 594.384,Z 495.448,A -85,B 0,C 180,E1 -1222.913,E2 -1222.913} C_VEL
LIN {X 0,Y 594.382,Z 495.44,A -85,B 0,C 180,E1 -1225.859,E2 -1225.859} C_VEL
LIN {X 0,Y 594.387,Z 495.447,A -85,B 0,C 180,E1 -1228.65,E2 -1228.65} C_VEL
LIN {X 0,Y 594.381,Z 495.447,A -85,B 0,C 180,E1 -1231.04,E2 -1231.04} C_VEL
LIN {X 0,Y 594.389,Z 495.439,A -85,B 0,C 180,E1 -1233.974,E2 -1233.974} C_VEL
LIN {X 0,Y 594.386,Z 495.441,A -85,B 0,C 180,E1 -1236.295,E2 -1236.295} C_VEL
LIN {X 0,Y 594.402,Z 495.442,A -85,B 0,C 180,E1 -1239.224,E2 -1239.224} C_VEL
LIN {X 0,Y 594.374,Z 495.441,A -85,B 0,C 180,E1 -1242.095,E2 -1242.095} C_VEL
LIN {X 0,Y 594.366,Z 495.443,A -85,B 0,C 180,E1 -1244.219,E2 -1244.219} C_VEL
LIN {X 0,Y 594.367,Z 495.451,A -85,B 0,C 180,E1 -1247.017,E2 -1247.017} C_VEL
LIN {X 0,Y 594.39,Z 495.439,A -85,B 0,C 180,E1 -1249.784,E2 -1249.784} C_VEL
LIN {X 0,Y 594.412,Z 495.44,A -85,B 0,C 180,E1 -1252.527,E2 -1252.527} C_VEL
LIN {X 0,Y 594.399,Z 495.444,A -85,B 0,C 180,E1 -1255.252,E2 -1255.252} C_VEL
LIN {X 0,Y 594.387,Z 495.439,A -85,B 0,C 180,E1 -1257.967,E2 -1257.967} C_VEL
LIN {X 0,Y 594.419,Z 495.44,A -85,B 0,C 180,E1 -1260.677,E2 -1260.677} C_VEL
LIN {X 0,Y 594.386,Z 495.444,A -85,B 0,C 180,E1 -1263.389,E2 -1263.389} C_VEL
LIN {X 0,Y 594.38,Z 495.44,A -85,B 0,C 180,E1 -1266.108,E2 -1266.108} C_VEL
LIN {X 0,Y 594.398,Z 495.445,A -85,B 0,C 180,E1 -1268.842,E2 -1268.842} C_VEL
LIN {X 0,Y 594.388,Z 495.442,A -85,B 0,C 180,E1 -1271.595,E2 -1271.595} C_VEL
LIN {X 0,Y 594.38,Z 495.441,A -85,B 0,C 180,E1 -1274.377,E2 -1274.377} C_VEL
LIN {X 0,Y 594.36,Z 495.448,A -85,B 0,C 180,E1 -1275.34,E2 -1275.34} C_VEL
LIN {X 0,Y 593.69,Z 495.528,A -85,B 0,C 180,E1 -1275.906,E2 -1275.906} C_VEL
LIN {X 0,Y 590.836,Z 495.887,A -85,B 0,C 180,E1 -1276.824,E2 -1276.824} C_VEL
LIN {X 0,Y 588.429,Z 496.185,A -85,B 0,C 180,E1 -1277.563,E2 -1277.563} C_VEL
LIN {X 0,Y 587.402,Z 496.31,A -85,B 0,C 180,E1 -1278.133,E2 -1278.133} C_VEL
LIN {X 0,Y 587.321,Z 496.32,A -85,B 0,C 180,E1 -1278.326,E2 -1278.326} C_VEL
LIN {X 0,Y 587.347,Z 496.326,A -85,B 0,C 180,E1 -1281.045,E2 -1281.045} C_VEL
LIN {X 0,Y 587.329,Z 496.319,A -85,B 0,C 180,E1 -1284.006,E2 -1284.006} C_VEL
LIN {X 0,Y 587.355,Z 496.316,A -85,B 0,C 180,E1 -1286.277,E2 -1286.277} C_VEL
LIN {X 0,Y 587.346,Z 496.327,A -85,B 0,C 180,E1 -1289.135,E2 -1289.135} C_VEL
LIN {X 0,Y 587.349,Z 496.319,A -85,B 0,C 180,E1 -1291.838,E2 -1291.838} C_VEL
LIN {X 0,Y 587.391,Z 496.442,A -85,B 0,C 180,E1 -1294.527,E2 -1294.527} C_VEL
LIN {X 0,Y 587.362,Z 509.295,A -85,B 0,C 180,E1 -1296.96,E2 -1296.96} C_VEL
LIN {X 0,Y 587.318,Z 517.873,A -85,B 0,C 180,E1 -1298.567,E2 -1298.567} C_VEL
LIN {X 0,Y 587.851,Z 523.059,A -85,B 0,C 180,E1 -1298.649,E2 -1298.649} C_VEL
LIN {X 0,Y 587.716,Z 624.541,A -85,B 0,C 180,E1 -1299.911,E2 -1299.911} C_VEL
LIN {X 0,Y 587.657,Z 637.922,A -85,B 0,C 180,E1 -1300.225,E2 -1300.225} C_VEL
LIN {X 0,Y 587.607,Z 650.893,A -85,B 0,C 180,E1 -1300.68,E2 -1300.68} C_VEL
LIN {X 0,Y 587.556,Z 662.82,A -85,B 0,C 180,E1 -1301.252,E2 -1301.252} C_VEL
LIN {X 0,Y 587.469,Z 674.154,A -85,B 0,C 180,E1 -1301.946,E2 -1301.946} C_VEL
LIN {X 0,Y 587.361,Z 684.859,A -85,B 0,C 180,E1 -1302.768,E2 -1302.768} C_VEL
LIN {X 0,Y 587.335,Z 694.834,A -85,B 0,C 180,E1 -1303.728,E2 -1303.728} C_VEL
LIN {X 0,Y 587.268,Z 703.5,A -85,B 0,C 180,E1 -1304.758,E2 -1304.758} C_VEL
LIN {X 0,Y 587.217,Z 711.077,A -85,B 0,C 180,E1 -1305.897,E2 -1305.897} C_VEL
LIN {X 0,Y 587.195,Z 716.783,A -85,B 0,C 180,E1 -1306.984,E2 -1306.984} C_VEL
LIN {X 0,Y 587.184,Z 720.631,A -85,B 0,C 180,E1 -1307.914,E2 -1307.914} C_VEL
LIN {X 0,Y 587.131,Z 723.902,A -85,B 0,C 180,E1 -1308.947,E2 -1308.947} C_VEL
LIN {X 0,Y 587.139,Z 726.225,A -85,B 0,C 180,E1 -1310.002,E2 -1310.002} C_VEL
LIN {X 0,Y 587.108,Z 727.597,A -85,B 0,C 180,E1 -1311.085,E2 -1311.085} C_VEL
LIN {X 0,Y 587.136,Z 727.931,A -85,B 0,C 180,E1 -1312.378,E2 -1312.378} C_VEL
LIN {X 0,Y 587.12,Z 727.293,A -85,B 0,C 180,E1 -1313.322,E2 -1313.322} C_VEL
LIN {X 0,Y 587.132,Z 725.461,A -85,B 0,C 180,E1 -1314.484,E2 -1314.484} C_VEL
LIN {X 0,Y 587.157,Z 722.058,A -85,B 0,C 180,E1 -1315.767,E2 -1315.767} C_VEL
LIN {X 0,Y 587.166,Z 717.682,A -85,B 0,C 180,E1 -1316.914,E2 -1316.914} C_VEL
LIN {X 0,Y 587.217,Z 712.071,A -85,B 0,C 180,E1 -1318.023,E2 -1318.023} C_VEL
LIN {X 0,Y 587.248,Z 705.678,A -85,B 0,C 180,E1 -1319.029,E2 -1319.029} C_VEL
LIN {X 0,Y 587.285,Z 697.868,A -85,B 0,C 180,E1 -1320.026,E2 -1320.026} C_VEL
LIN {X 0,Y 587.352,Z 689.177,A -85,B 0,C 180,E1 -1320.933,E2 -1320.933} C_VEL
LIN {X 0,Y 587.407,Z 678.945,A -85,B 0,C 180,E1 -1321.798,E2 -1321.798} C_VEL
LIN {X 0,Y 587.497,Z 667.411,A -85,B 0,C 180,E1 -1322.577,E2 -1322.577} C_VEL
LIN {X 0,Y 587.557,Z 655.545,A -85,B 0,C 180,E1 -1323.206,E2 -1323.206} C_VEL
LIN {X 0,Y 587.651,Z 643.436,A -85,B 0,C 180,E1 -1323.689,E2 -1323.689} C_VEL
LIN {X 0,Y 587.689,Z 630.872,A -85,B 0,C 180,E1 -1324.049,E2 -1324.049} C_VEL
LIN {X 0,Y 587.742,Z 618.896,A -85,B 0,C 180,E1 -1324.266,E2 -1324.266} C_VEL
LIN {X 0,Y 587.795,Z 520.768,A -85,B 0,C 180,E1 -1325.471,E2 -1325.471} C_VEL
LIN {X 0,Y 587.323,Z 517.838,A -85,B 0,C 180,E1 -1325.529,E2 -1325.529} C_VEL
LIN {X 0,Y 587.39,Z 503.47,A -85,B 0,C 180,E1 -1328.229,E2 -1328.229} C_VEL
LIN {X 0,Y 587.351,Z 496.319,A -85,B 0,C 180,E1 -1329.605,E2 -1329.605} C_VEL
LIN {X 0,Y 587.354,Z 496.322,A -85,B 0,C 180,E1 -1332.595,E2 -1332.595} C_VEL
LIN {X 0,Y 587.362,Z 496.314,A -85,B 0,C 180,E1 -1335.74,E2 -1335.74} C_VEL
LIN {X 0,Y 587.345,Z 496.327,A -85,B 0,C 180,E1 -1338.867,E2 -1338.867} C_VEL
LIN {X 0,Y 587.363,Z 496.314,A -85,B 0,C 180,E1 -1341.745,E2 -1341.745} C_VEL
LIN {X 0,Y 587.363,Z 496.318,A -85,B 0,C 180,E1 -1344.507,E2 -1344.507} C_VEL
LIN {X 0,Y 587.369,Z 496.318,A -85,B 0,C 180,E1 -1347.257,E2 -1347.257} C_VEL
LIN {X 0,Y 587.383,Z 496.312,A -85,B 0,C 180,E1 -1350,E2 -1350} C_VEL
LIN {X 0,Y 587.371,Z 496.321,A -85,B 0,C 180,E1 -1352.743,E2 -1352.743} C_VEL
LIN {X 0,Y 587.36,Z 496.317,A -85,B 0,C 180,E1 -1355.493,E2 -1355.493} C_VEL
LIN {X 0,Y 587.368,Z 496.315,A -85,B 0,C 180,E1 -1358.255,E2 -1358.255} C_VEL
LIN {X 0,Y 587.345,Z 496.324,A -85,B 0,C 180,E1 -1361.133,E2 -1361.133} C_VEL
LIN {X 0,Y 587.362,Z 496.315,A -85,B 0,C 180,E1 -1364.26,E2 -1364.26} C_VEL
LIN {X 0,Y 587.355,Z 496.319,A -85,B 0,C 180,E1 -1367.405,E2 -1367.405} C_VEL
LIN {X 0,Y 587.328,Z 496.32,A -85,B 0,C 180,E1 -1370.304,E2 -1370.304} C_VEL
LIN {X 0,Y 587.319,Z 496.326,A -85,B 0,C 180,E1 -1373.258,E2 -1373.258} C_VEL
LIN {X 0,Y 587.331,Z 496.321,A -85,B 0,C 180,E1 -1375.516,E2 -1375.516} C_VEL
LIN {X 0,Y 587.345,Z 496.317,A -85,B 0,C 180,E1 -1377.817,E2 -1377.817} C_VEL
LIN {X 0,Y 587.347,Z 496.319,A -85,B 0,C 180,E1 -1380.512,E2 -1380.512} C_VEL
LIN {X 0,Y 587.33,Z 496.323,A -85,B 0,C 180,E1 -1383.396,E2 -1383.396} C_VEL
LIN {X 0,Y 587.35,Z 496.316,A -85,B 0,C 180,E1 -1385.895,E2 -1385.895} C_VEL
LIN {X 0,Y 587.33,Z 496.32,A -85,B 0,C 180,E1 -1388.478,E2 -1388.478} C_VEL
LIN {X 0,Y 587.357,Z 496.324,A -85,B 0,C 180,E1 -1391.154,E2 -1391.154} C_VEL
LIN {X 0,Y 587.326,Z 496.319,A -85,B 0,C 180,E1 -1394.114,E2 -1394.114} C_VEL
LIN {X 0,Y 587.315,Z 496.33,A -85,B 0,C 180,E1 -1396.994,E2 -1396.994} C_VEL
LIN {X 0,Y 587.314,Z 496.321,A -85,B 0,C 180,E1 -1399.746,E2 -1399.746} C_VEL
LIN {X 0,Y 587.338,Z 496.318,A -85,B 0,C 180,E1 -1402.392,E2 -1402.392} C_VEL
LIN {X 0,Y 587.347,Z 496.324,A -85,B 0,C 180,E1 -1404.946,E2 -1404.946} C_VEL
LIN {X 0,Y 587.333,Z 496.323,A -85,B 0,C 180,E1 -1407.421,E2 -1407.421} C_VEL
LIN {X 0,Y 587.338,Z 496.318,A -85,B 0,C 180,E1 -1409.831,E2 -1409.831} C_VEL
LIN {X 0,Y 587.341,Z 496.317,A -85,B 0,C 180,E1 -1412.307,E2 -1412.307} C_VEL
LIN {X 0,Y 587.335,Z 496.319,A -85,B 0,C 180,E1 -1414.484,E2 -1414.484} C_VEL
LIN {X 0,Y 587.333,Z 496.323,A -85,B 0,C 180,E1 -1417.486,E2 -1417.486} C_VEL
LIN {X 0,Y 587.327,Z 496.321,A -85,B 0,C 180,E1 -1419.695,E2 -1419.695} C_VEL
LIN {X 0,Y 587.352,Z 496.318,A -85,B 0,C 180,E1 -1422.594,E2 -1422.594} C_VEL
LIN {X 0,Y 587.354,Z 496.317,A -85,B 0,C 180,E1 -1425.739,E2 -1425.739} C_VEL
LIN {X 0,Y 587.351,Z 496.321,A -85,B 0,C 180,E1 -1428.859,E2 -1428.859} C_VEL
LIN {X 0,Y 587.364,Z 496.316,A -85,B 0,C 180,E1 -1431.745,E2 -1431.745} C_VEL
LIN {X 0,Y 587.358,Z 496.316,A -85,B 0,C 180,E1 -1434.507,E2 -1434.507} C_VEL
LIN {X 0,Y 587.378,Z 496.322,A -85,B 0,C 180,E1 -1437.257,E2 -1437.257} C_VEL
LIN {X 0,Y 587.373,Z 496.313,A -85,B 0,C 180,E1 -1440,E2 -1440} C_VEL
LIN {X 0,Y 587.377,Z 496.315,A -85,B 0,C 180,E1 -1442.744,E2 -1442.744} C_VEL
LIN {X 0,Y 587.364,Z 496.32,A -85,B 0,C 180,E1 -1445.493,E2 -1445.493} C_VEL
LIN {X 0,Y 587.365,Z 496.314,A -85,B 0,C 180,E1 -1448.256,E2 -1448.256} C_VEL
LIN {X 0,Y 587.352,Z 496.325,A -85,B 0,C 180,E1 -1451.142,E2 -1451.142} C_VEL
LIN {X 0,Y 587.355,Z 496.315,A -85,B 0,C 180,E1 -1454.262,E2 -1454.262} C_VEL
LIN {X 0,Y 587.355,Z 496.323,A -85,B 0,C 180,E1 -1457.406,E2 -1457.406} C_VEL
LIN {X 0,Y 587.328,Z 496.318,A -85,B 0,C 180,E1 -1460.305,E2 -1460.305} C_VEL
LIN {X 0,Y 587.317,Z 496.331,A -85,B 0,C 180,E1 -1463.259,E2 -1463.259} C_VEL
LIN {X 0,Y 587.356,Z 496.315,A -85,B 0,C 180,E1 -1466.183,E2 -1466.183} C_VEL
LIN {X 0,Y 587.347,Z 496.324,A -85,B 0,C 180,E1 -1469.135,E2 -1469.135} C_VEL
LIN {X 0,Y 587.35,Z 496.318,A -85,B 0,C 180,E1 -1471.839,E2 -1471.839} C_VEL
LIN {X 0,Y 587.353,Z 496.315,A -85,B 0,C 180,E1 -1474.35,E2 -1474.35} C_VEL
LIN {X 0,Y 587.348,Z 496.318,A -85,B 0,C 180,E1 -1476.747,E2 -1476.747} C_VEL
LIN {X 0,Y 587.344,Z 496.327,A -85,B 0,C 180,E1 -1479.36,E2 -1479.36} C_VEL
LIN {X 0,Y 587.33,Z 496.319,A -85,B 0,C 180,E1 -1482.109,E2 -1482.109} C_VEL
LIN {X 0,Y 587.312,Z 496.327,A -85,B 0,C 180,E1 -1485.09,E2 -1485.09} C_VEL
LIN {X 0,Y 587.35,Z 496.318,A -85,B 0,C 180,E1 -1487.928,E2 -1487.928} C_VEL
LIN {X 0,Y 587.334,Z 496.323,A -85,B 0,C 180,E1 -1491.059,E2 -1491.059} C_VEL
LIN {X 0,Y 587.351,Z 496.325,A -85,B 0,C 180,E1 -1493.293,E2 -1493.293} C_VEL
LIN {X 0,Y 587.363,Z 496.319,A -85,B 0,C 180,E1 -1495.781,E2 -1495.781} C_VEL
LIN {X 0,Y 587.352,Z 496.316,A -85,B 0,C 180,E1 -1498.233,E2 -1498.233} C_VEL
LIN {X 0,Y 587.349,Z 496.319,A -85,B 0,C 180,E1 -1500.867,E2 -1500.867} C_VEL
LIN {X 0,Y 587.358,Z 496.321,A -85,B 0,C 180,E1 -1503.82,E2 -1503.82} C_VEL
LIN {X 0,Y 587.406,Z 496.46,A -85,B 0,C 180,E1 -1506.021,E2 -1506.021} C_VEL
LIN {X 0,Y 587.992,Z 500.383,A -85,B 0,C 180,E1 -1506.584,E2 -1506.584} C_VEL
LIN {X 0,Y 587.783,Z 522.219,A -85,B 0,C 180,E1 -1509.529,E2 -1509.529} C_VEL
LIN {X 0,Y 587.62,Z 542.689,A -85,B 0,C 180,E1 -1512.243,E2 -1512.243} C_VEL
LIN {X 0,Y 587.474,Z 563.16,A -85,B 0,C 180,E1 -1514.919,E2 -1514.919} C_VEL
LIN {X 0,Y 587.418,Z 575.357,A -85,B 0,C 180,E1 -1516.498,E2 -1516.498} C_VEL
LIN {X 0,Y 587.891,Z 579.746,A -85,B 0,C 180,E1 -1516.564,E2 -1516.564} C_VEL
LIN {X 0,Y 587.715,Z 683.962,A -85,B 0,C 180,E1 -1517.855,E2 -1517.855} C_VEL
LIN {X 0,Y 587.666,Z 697.228,A -85,B 0,C 180,E1 -1518.161,E2 -1518.161} C_VEL
LIN {X 0,Y 587.614,Z 710.104,A -85,B 0,C 180,E1 -1518.604,E2 -1518.604} C_VEL
LIN {X 0,Y 587.554,Z 721.636,A -85,B 0,C 180,E1 -1519.141,E2 -1519.141} C_VEL
LIN {X 0,Y 587.458,Z 733.204,A -85,B 0,C 180,E1 -1519.837,E2 -1519.837} C_VEL
LIN {X 0,Y 587.391,Z 743.6,A -85,B 0,C 180,E1 -1520.618,E2 -1520.618} C_VEL
LIN {X 0,Y 587.321,Z 752.114,A -85,B 0,C 180,E1 -1521.398,E2 -1521.398} C_VEL
LIN {X 0,Y 587.274,Z 759.962,A -85,B 0,C 180,E1 -1522.263,E2 -1522.263} C_VEL
LIN {X 0,Y 587.23,Z 766.471,A -85,B 0,C 180,E1 -1523.127,E2 -1523.127} C_VEL
LIN {X 0,Y 587.236,Z 772.867,A -85,B 0,C 180,E1 -1524.161,E2 -1524.161} C_VEL
LIN {X 0,Y 587.147,Z 777.95,A -85,B 0,C 180,E1 -1525.194,E2 -1525.194} C_VEL
LIN {X 0,Y 587.212,Z 781.896,A -85,B 0,C 180,E1 -1526.226,E2 -1526.226} C_VEL
LIN {X 0,Y 587.132,Z 784.809,A -85,B 0,C 180,E1 -1527.256,E2 -1527.256} C_VEL
LIN {X 0,Y 587.138,Z 786.201,A -85,B 0,C 180,E1 -1527.942,E2 -1527.942} C_VEL
LIN {X 0,Y 587.14,Z 787.784,A -85,B 0,C 180,E1 -1529.314,E2 -1529.314} C_VEL
LIN {X 0,Y 587.137,Z 788,A -85,B 0,C 180,E1 -1530,E2 -1530} C_VEL
LIN {X 0,Y 587.147,Z 787.185,A -85,B 0,C 180,E1 -1531.372,E2 -1531.372} C_VEL
LIN {X 0,Y 587.138,Z 786.201,A -85,B 0,C 180,E1 -1532.058,E2 -1532.058} C_VEL
LIN {X 0,Y 587.132,Z 784.81,A -85,B 0,C 180,E1 -1532.744,E2 -1532.744} C_VEL
LIN {X 0,Y 587.212,Z 781.896,A -85,B 0,C 180,E1 -1533.774,E2 -1533.774} C_VEL
LIN {X 0,Y 587.147,Z 777.95,A -85,B 0,C 180,E1 -1534.806,E2 -1534.806} C_VEL
LIN {X 0,Y 587.217,Z 771.878,A -85,B 0,C 180,E1 -1536.011,E2 -1536.011} C_VEL
LIN {X 0,Y 587.245,Z 765.238,A -85,B 0,C 180,E1 -1537.046,E2 -1537.046} C_VEL
LIN {X 0,Y 587.299,Z 756.992,A -85,B 0,C 180,E1 -1538.083,E2 -1538.083} C_VEL
LIN {X 0,Y 587.343,Z 748.54,A -85,B 0,C 180,E1 -1538.949,E2 -1538.949} C_VEL
LIN {X 0,Y 587.41,Z 738.098,A -85,B 0,C 180,E1 -1539.816,E2 -1539.816} C_VEL
LIN {X 0,Y 587.505,Z 727.763,A -85,B 0,C 180,E1 -1540.511,E2 -1540.511} C_VEL
LIN {X 0,Y 587.584,Z 715.807,A -85,B 0,C 180,E1 -1541.149,E2 -1541.149} C_VEL
LIN {X 0,Y 587.624,Z 703.599,A -85,B 0,C 180,E1 -1541.639,E2 -1541.639} C_VEL
LIN {X 0,Y 587.683,Z 690.448,A -85,B 0,C 180,E1 -1542.014,E2 -1542.014} C_VEL
LIN {X 0,Y 587.771,Z 678.106,A -85,B 0,C 180,E1 -1542.231,E2 -1542.231} C_VEL
LIN {X 0,Y 587.743,Z 577.51,A -85,B 0,C 180,E1 -1543.467,E2 -1543.467} C_VEL
LIN {X 0,Y 587.424,Z 575.272,A -85,B 0,C 180,E1 -1543.513,E2 -1543.513} C_VEL
LIN {X 0,Y 587.569,Z 553.607,A -85,B 0,C 180,E1 -1546.325,E2 -1546.325} C_VEL
LIN {X 0,Y 587.736,Z 531.097,A -85,B 0,C 180,E1 -1549.287,E2 -1549.287} C_VEL
LIN {X 0,Y 587.893,Z 508.571,A -85,B 0,C 180,E1 -1552.306,E2 -1552.306} C_VEL
LIN {X 0,Y 587.877,Z 499.018,A -85,B 0,C 180,E1 -1553.608,E2 -1553.608} C_VEL
LIN {X 0,Y 587.365,Z 496.322,A -85,B 0,C 180,E1 -1554.005,E2 -1554.005} C_VEL
LIN {X 0,Y 587.331,Z 496.323,A -85,B 0,C 180,E1 -1557.045,E2 -1557.045} C_VEL
LIN {X 0,Y 587.346,Z 496.318,A -85,B 0,C 180,E1 -1559.379,E2 -1559.379} C_VEL
LIN {X 0,Y 587.355,Z 496.316,A -85,B 0,C 180,E1 -1561.837,E2 -1561.837} C_VEL
LIN {X 0,Y 587.355,Z 496.321,A -85,B 0,C 180,E1 -1564.348,E2 -1564.348} C_VEL
LIN {X 0,Y 587.353,Z 496.325,A -85,B 0,C 180,E1 -1566.746,E2 -1566.746} C_VEL
LIN {X 0,Y 587.344,Z 496.318,A -85,B 0,C 180,E1 -1569.358,E2 -1569.358} C_VEL
LIN {X 0,Y 587.334,Z 496.32,A -85,B 0,C 180,E1 -1572.107,E2 -1572.107} C_VEL
LIN {X 0,Y 587.312,Z 496.325,A -85,B 0,C 180,E1 -1575.088,E2 -1575.088} C_VEL
LIN {X 0,Y 587.348,Z 496.316,A -85,B 0,C 180,E1 -1577.927,E2 -1577.927} C_VEL
LIN {X 0,Y 587.332,Z 496.324,A -85,B 0,C 180,E1 -1581.057,E2 -1581.057} C_VEL
LIN {X 0,Y 587.35,Z 496.318,A -85,B 0,C 180,E1 -1583.29,E2 -1583.29} C_VEL
LIN {X 0,Y 587.365,Z 496.314,A -85,B 0,C 180,E1 -1585.78,E2 -1585.78} C_VEL
LIN {X 0,Y 587.348,Z 496.318,A -85,B 0,C 180,E1 -1588.231,E2 -1588.231} C_VEL
LIN {X 0,Y 587.347,Z 496.326,A -85,B 0,C 180,E1 -1590.865,E2 -1590.865} C_VEL
LIN {X 0,Y 587.357,Z 496.315,A -85,B 0,C 180,E1 -1593.817,E2 -1593.817} C_VEL
LIN {X 0,Y 587.317,Z 496.328,A -85,B 0,C 180,E1 -1596.741,E2 -1596.741} C_VEL
LIN {X 0,Y 587.327,Z 496.319,A -85,B 0,C 180,E1 -1599.695,E2 -1599.695} C_VEL
LIN {X 0,Y 587.351,Z 496.321,A -85,B 0,C 180,E1 -1602.594,E2 -1602.594} C_VEL
LIN {X 0,Y 587.355,Z 496.315,A -85,B 0,C 180,E1 -1605.739,E2 -1605.739} C_VEL
LIN {X 0,Y 587.352,Z 496.325,A -85,B 0,C 180,E1 -1608.858,E2 -1608.858} C_VEL
LIN {X 0,Y 587.364,Z 496.315,A -85,B 0,C 180,E1 -1611.744,E2 -1611.744} C_VEL
LIN {X 0,Y 587.358,Z 496.318,A -85,B 0,C 180,E1 -1614.507,E2 -1614.507} C_VEL
LIN {X 0,Y 587.377,Z 496.319,A -85,B 0,C 180,E1 -1617.256,E2 -1617.256} C_VEL
LIN {X 0,Y 587.373,Z 496.313,A -85,B 0,C 180,E1 -1620,E2 -1620} C_VEL
LIN {X 0,Y 587.376,Z 496.318,A -85,B 0,C 180,E1 -1622.743,E2 -1622.743} C_VEL
LIN {X 0,Y 587.362,Z 496.318,A -85,B 0,C 180,E1 -1625.493,E2 -1625.493} C_VEL
LIN {X 0,Y 587.364,Z 496.315,A -85,B 0,C 180,E1 -1628.255,E2 -1628.255} C_VEL
LIN {X 0,Y 587.351,Z 496.326,A -85,B 0,C 180,E1 -1631.141,E2 -1631.141} C_VEL
LIN {X 0,Y 587.354,Z 496.316,A -85,B 0,C 180,E1 -1634.261,E2 -1634.261} C_VEL
LIN {X 0,Y 587.353,Z 496.322,A -85,B 0,C 180,E1 -1637.405,E2 -1637.405} C_VEL
LIN {X 0,Y 587.321,Z 496.32,A -85,B 0,C 180,E1 -1638.326,E2 -1638.326} C_VEL
LIN {X 0,Y 586.668,Z 496.409,A -85,B 0,C 180,E1 -1638.898,E2 -1638.898} C_VEL
LIN {X 0,Y 583.835,Z 496.767,A -85,B 0,C 180,E1 -1639.826,E2 -1639.826} C_VEL
LIN {X 0,Y 581.425,Z 497.069,A -85,B 0,C 180,E1 -1640.573,E2 -1640.573} C_VEL
LIN {X 0,Y 580.372,Z 497.196,A -85,B 0,C 180,E1 -1641.149,E2 -1641.149} C_VEL
LIN {X 0,Y 580.278,Z 497.205,A -85,B 0,C 180,E1 -1641.345,E2 -1641.345} C_VEL
LIN {X 0,Y 580.291,Z 497.196,A -85,B 0,C 180,E1 -1644.316,E2 -1644.316} C_VEL
LIN {X 0,Y 580.302,Z 497.197,A -85,B 0,C 180,E1 -1646.622,E2 -1646.622} C_VEL
LIN {X 0,Y 580.3,Z 497.204,A -85,B 0,C 180,E1 -1649.312,E2 -1649.312} C_VEL
LIN {X 0,Y 580.295,Z 497.196,A -85,B 0,C 180,E1 -1652.2,E2 -1652.2} C_VEL
LIN {X 0,Y 580.337,Z 497.308,A -85,B 0,C 180,E1 -1654.474,E2 -1654.474} C_VEL
LIN {X 0,Y 580.341,Z 510.181,A -85,B 0,C 180,E1 -1656.942,E2 -1656.942} C_VEL
LIN {X 0,Y 580.268,Z 517.85,A -85,B 0,C 180,E1 -1658.396,E2 -1658.396} C_VEL
LIN {X 0,Y 580.961,Z 523.634,A -85,B 0,C 180,E1 -1658.494,E2 -1658.494} C_VEL
LIN {X 0,Y 580.804,Z 624.121,A -85,B 0,C 180,E1 -1659.757,E2 -1659.757} C_VEL
LIN {X 0,Y 580.711,Z 637.365,A -85,B 0,C 180,E1 -1660.066,E2 -1660.066} C_VEL
LIN {X 0,Y 580.647,Z 649.92,A -85,B 0,C 180,E1 -1660.503,E2 -1660.503} C_VEL
LIN {X 0,Y 580.547,Z 661.116,A -85,B 0,C 180,E1 -1661.025,E2 -1661.025} C_VEL
LIN {X 0,Y 580.467,Z 673.117,A -85,B 0,C 180,E1 -1661.752,E2 -1661.752} C_VEL
LIN {X 0,Y 580.32,Z 684.334,A -85,B 0,C 180,E1 -1662.609,E2 -1662.609} C_VEL
LIN {X 0,Y 580.282,Z 693.641,A -85,B 0,C 180,E1 -1663.497,E2 -1663.497} C_VEL
LIN {X 0,Y 580.2,Z 701.312,A -85,B 0,C 180,E1 -1664.385,E2 -1664.385} C_VEL
LIN {X 0,Y 580.17,Z 708.286,A -85,B 0,C 180,E1 -1665.366,E2 -1665.366} C_VEL
LIN {X 0,Y 580.113,Z 713.873,A -85,B 0,C 180,E1 -1666.328,E2 -1666.328} C_VEL
LIN {X 0,Y 580.095,Z 718.351,A -85,B 0,C 180,E1 -1667.278,E2 -1667.278} C_VEL
LIN {X 0,Y 580.095,Z 721.87,A -85,B 0,C 180,E1 -1668.216,E2 -1668.216} C_VEL
LIN {X 0,Y 580.025,Z 724.475,A -85,B 0,C 180,E1 -1669.134,E2 -1669.134} C_VEL
LIN {X 0,Y 580.045,Z 726.339,A -85,B 0,C 180,E1 -1670.048,E2 -1670.048} C_VEL
LIN {X 0,Y 580.007,Z 727.503,A -85,B 0,C 180,E1 -1670.944,E2 -1670.944} C_VEL
LIN {X 0,Y 580.014,Z 727.987,A -85,B 0,C 180,E1 -1671.961,E2 -1671.961} C_VEL
LIN {X 0,Y 580.026,Z 727.538,A -85,B 0,C 180,E1 -1673.101,E2 -1673.101} C_VEL
LIN {X 0,Y 580.041,Z 725.616,A -85,B 0,C 180,E1 -1674.439,E2 -1674.439} C_VEL
LIN {X 0,Y 580.068,Z 723.091,A -85,B 0,C 180,E1 -1675.474,E2 -1675.474} C_VEL
LIN {X 0,Y 580.087,Z 718.744,A -85,B 0,C 180,E1 -1676.716,E2 -1676.716} C_VEL
LIN {X 0,Y 580.143,Z 713.723,A -85,B 0,C 180,E1 -1677.791,E2 -1677.791} C_VEL
LIN {X 0,Y 580.18,Z 706.523,A -85,B 0,C 180,E1 -1678.995,E2 -1678.995} C_VEL
LIN {X 0,Y 580.226,Z 698.711,A -85,B 0,C 180,E1 -1680.025,E2 -1680.025} C_VEL
LIN {X 0,Y 580.312,Z 689.342,A -85,B 0,C 180,E1 -1681.026,E2 -1681.026} C_VEL
LIN {X 0,Y 580.394,Z 679.016,A -85,B 0,C 180,E1 -1681.912,E2 -1681.912} C_VEL
LIN {X 0,Y 580.499,Z 667.386,A -85,B 0,C 180,E1 -1682.707,E2 -1682.707} C_VEL
LIN {X 0,Y 580.594,Z 655.482,A -85,B 0,C 180,E1 -1683.345,E2 -1683.345} C_VEL
LIN {X 0,Y 580.67,Z 643.166,A -85,B 0,C 180,E1 -1683.841,E2 -1683.841} C_VEL
LIN {X 0,Y 580.746,Z 629.763,A -85,B 0,C 180,E1 -1684.221,E2 -1684.221} C_VEL
LIN {X 0,Y 580.811,Z 615.882,A -85,B 0,C 180,E1 -1684.453,E2 -1684.453} C_VEL
LIN {X 0,Y 580.815,Z 521.268,A -85,B 0,C 180,E1 -1685.629,E2 -1685.629} C_VEL
LIN {X 0,Y 580.284,Z 517.908,A -85,B 0,C 180,E1 -1685.684,E2 -1685.684} C_VEL
LIN {X 0,Y 580.367,Z 504.016,A -85,B 0,C 180,E1 -1688.326,E2 -1688.326} C_VEL
LIN {X 0,Y 580.296,Z 497.198,A -85,B 0,C 180,E1 -1689.67,E2 -1689.67} C_VEL
LIN {X 0,Y 580.3,Z 497.198,A -85,B 0,C 180,E1 -1692.376,E2 -1692.376} C_VEL
LIN {X 0,Y 580.284,Z 497.2,A -85,B 0,C 180,E1 -1695.266,E2 -1695.266} C_VEL
LIN {X 0,Y 580.307,Z 497.194,A -85,B 0,C 180,E1 -1698.119,E2 -1698.119} C_VEL
LIN {X 0,Y 580.278,Z 497.207,A -85,B 0,C 180,E1 -1700.941,E2 -1700.941} C_VEL
LIN {X 0,Y 580.309,Z 497.197,A -85,B 0,C 180,E1 -1703.254,E2 -1703.254} C_VEL
LIN {X 0,Y 580.272,Z 497.198,A -85,B 0,C 180,E1 -1705.833,E2 -1705.833} C_VEL
LIN {X 0,Y 580.342,Z 497.189,A -85,B 0,C 180,E1 -1707.918,E2 -1707.918} C_VEL
LIN {X 0,Y 580.361,Z 497.193,A -85,B 0,C 180,E1 -1710.694,E2 -1710.694} C_VEL
LIN {X 0,Y 580.282,Z 497.199,A -85,B 0,C 180,E1 -1713.472,E2 -1713.472} C_VEL
LIN {X 0,Y 580.327,Z 497.192,A -85,B 0,C 180,E1 -1715.56,E2 -1715.56} C_VEL
LIN {X 0,Y 580.331,Z 497.192,A -85,B 0,C 180,E1 -1718.356,E2 -1718.356} C_VEL
LIN {X 0,Y 580.297,Z 497.201,A -85,B 0,C 180,E1 -1721.191,E2 -1721.191} C_VEL
LIN {X 0,Y 580.324,Z 497.191,A -85,B 0,C 180,E1 -1724.017,E2 -1724.017} C_VEL
LIN {X 0,Y 580.308,Z 497.203,A -85,B 0,C 180,E1 -1726.913,E2 -1726.913} C_VEL
LIN {X 0,Y 580.303,Z 497.194,A -85,B 0,C 180,E1 -1729.822,E2 -1729.822} C_VEL
LIN {X 0,Y 580.291,Z 497.202,A -85,B 0,C 180,E1 -1732.802,E2 -1732.802} C_VEL
LIN {X 0,Y 580.303,Z 497.203,A -85,B 0,C 180,E1 -1735.079,E2 -1735.079} C_VEL
LIN {X 0,Y 580.297,Z 497.195,A -85,B 0,C 180,E1 -1738.185,E2 -1738.185} C_VEL
LIN {X 0,Y 580.296,Z 497.2,A -85,B 0,C 180,E1 -1740.697,E2 -1740.697} C_VEL
LIN {X 0,Y 580.299,Z 497.2,A -85,B 0,C 180,E1 -1743.316,E2 -1743.316} C_VEL
LIN {X 0,Y 580.319,Z 497.192,A -85,B 0,C 180,E1 -1745.767,E2 -1745.767} C_VEL
LIN {X 0,Y 580.284,Z 497.196,A -85,B 0,C 180,E1 -1748.146,E2 -1748.146} C_VEL
LIN {X 0,Y 580.314,Z 497.199,A -85,B 0,C 180,E1 -1750.841,E2 -1750.841} C_VEL
LIN {X 0,Y 580.283,Z 497.198,A -85,B 0,C 180,E1 -1753.656,E2 -1753.656} C_VEL
LIN {X 0,Y 580.277,Z 497.2,A -85,B 0,C 180,E1 -1756.608,E2 -1756.608} C_VEL
LIN {X 0,Y 580.294,Z 497.204,A -85,B 0,C 180,E1 -1759.157,E2 -1759.157} C_VEL
LIN {X 0,Y 580.283,Z 497.196,A -85,B 0,C 180,E1 -1761.926,E2 -1761.926} C_VEL
LIN {X 0,Y 580.302,Z 497.195,A -85,B 0,C 180,E1 -1764.457,E2 -1764.457} C_VEL
LIN {X 0,Y 580.284,Z 497.204,A -85,B 0,C 180,E1 -1766.975,E2 -1766.975} C_VEL
LIN {X 0,Y 580.301,Z 497.199,A -85,B 0,C 180,E1 -1769.426,E2 -1769.426} C_VEL
LIN {X 0,Y 580.31,Z 497.193,A -85,B 0,C 180,E1 -1772.137,E2 -1772.137} C_VEL
LIN {X 0,Y 580.302,Z 497.201,A -85,B 0,C 180,E1 -1774.92,E2 -1774.92} C_VEL
LIN {X 0,Y 580.267,Z 497.199,A -85,B 0,C 180,E1 -1777.948,E2 -1777.948} C_VEL
LIN {X 0,Y 580.307,Z 497.2,A -85,B 0,C 180,E1 -1780.914,E2 -1780.914} C_VEL
LIN {X 0,Y 580.275,Z 497.198,A -85,B 0,C 180,E1 -1783.826,E2 -1783.826} C_VEL
LIN {X 0,Y 580.273,Z 497.201,A -85,B 0,C 180,E1 -1786.696,E2 -1786.696} C_VEL
LIN {X 0,Y 580.298,Z 497.199,A -85,B 0,C 180,E1 -1789.534,E2 -1789.534} C_VEL
LIN {X 0,Y 580.332,Z 497.19,A -85,B 0,C 180,E1 -1792.345,E2 -1792.345} C_VEL
LIN {X 0,Y 580.338,Z 497.199,A -85,B 0,C 180,E1 -1795.137,E2 -1795.137} C_VEL
LIN {X 0,Y 580.329,Z 497.191,A -85,B 0,C 180,E1 -1797.918,E2 -1797.918} C_VEL
LIN {X 0,Y 580.36,Z 497.189,A -85,B 0,C 180,E1 -1800.694,E2 -1800.694} C_VEL
LIN {X 0,Y 580.288,Z 497.202,A -85,B 0,C 180,E1 -1803.472,E2 -1803.472} C_VEL
LIN {X 0,Y 580.33,Z 497.195,A -85,B 0,C 180,E1 -1805.56,E2 -1805.56} C_VEL
LIN {X 0,Y 580.329,Z 497.191,A -85,B 0,C 180,E1 -1808.356,E2 -1808.356} C_VEL
LIN {X 0,Y 580.323,Z 497.201,A -85,B 0,C 180,E1 -1811.209,E2 -1811.209} C_VEL
LIN {X 0,Y 580.319,Z 497.192,A -85,B 0,C 180,E1 -1814.017,E2 -1814.017} C_VEL
LIN {X 0,Y 580.306,Z 497.198,A -85,B 0,C 180,E1 -1816.916,E2 -1816.916} C_VEL
LIN {X 0,Y 580.301,Z 497.196,A -85,B 0,C 180,E1 -1819.823,E2 -1819.823} C_VEL
LIN {X 0,Y 580.269,Z 497.198,A -85,B 0,C 180,E1 -1822.053,E2 -1822.053} C_VEL
LIN {X 0,Y 580.303,Z 497.201,A -85,B 0,C 180,E1 -1825.08,E2 -1825.08} C_VEL
LIN {X 0,Y 580.313,Z 497.194,A -85,B 0,C 180,E1 -1827.864,E2 -1827.864} C_VEL
LIN {X 0,Y 580.293,Z 497.197,A -85,B 0,C 180,E1 -1830.698,E2 -1830.698} C_VEL
LIN {X 0,Y 580.299,Z 497.205,A -85,B 0,C 180,E1 -1833.318,E2 -1833.318} C_VEL
LIN {X 0,Y 580.322,Z 497.195,A -85,B 0,C 180,E1 -1835.769,E2 -1835.769} C_VEL
LIN {X 0,Y 580.284,Z 497.196,A -85,B 0,C 180,E1 -1838.147,E2 -1838.147} C_VEL
LIN {X 0,Y 580.297,Z 497.197,A -85,B 0,C 180,E1 -1840.844,E2 -1840.844} C_VEL
LIN {X 0,Y 580.284,Z 497.201,A -85,B 0,C 180,E1 -1843.658,E2 -1843.658} C_VEL
LIN {X 0,Y 580.289,Z 497.196,A -85,B 0,C 180,E1 -1846.609,E2 -1846.609} C_VEL
LIN {X 0,Y 580.299,Z 497.201,A -85,B 0,C 180,E1 -1849.158,E2 -1849.158} C_VEL
LIN {X 0,Y 580.29,Z 497.197,A -85,B 0,C 180,E1 -1851.928,E2 -1851.928} C_VEL
LIN {X 0,Y 580.284,Z 497.196,A -85,B 0,C 180,E1 -1854.456,E2 -1854.456} C_VEL
LIN {X 0,Y 580.291,Z 497.199,A -85,B 0,C 180,E1 -1856.976,E2 -1856.976} C_VEL
LIN {X 0,Y 580.304,Z 497.204,A -85,B 0,C 180,E1 -1859.426,E2 -1859.426} C_VEL
LIN {X 0,Y 580.298,Z 497.196,A -85,B 0,C 180,E1 -1862.142,E2 -1862.142} C_VEL
LIN {X 0,Y 580.323,Z 497.202,A -85,B 0,C 180,E1 -1865.27,E2 -1865.27} C_VEL
LIN {X 0,Y 580.344,Z 497.313,A -85,B 0,C 180,E1 -1865.829,E2 -1865.829} C_VEL
LIN {X 0,Y 581.106,Z 501.748,A -85,B 0,C 180,E1 -1866.478,E2 -1866.478} C_VEL
LIN {X 0,Y 580.881,Z 522.219,A -85,B 0,C 180,E1 -1869.275,E2 -1869.275} C_VEL
LIN {X 0,Y 580.682,Z 542.689,A -85,B 0,C 180,E1 -1872.024,E2 -1872.024} C_VEL
LIN {X 0,Y 580.497,Z 563.16,A -85,B 0,C 180,E1 -1874.733,E2 -1874.733} C_VEL
LIN {X 0,Y 580.435,Z 575.357,A -85,B 0,C 180,E1 -1876.332,E2 -1876.332} C_VEL
LIN {X 0,Y 580.972,Z 581.535,A -85,B 0,C 180,E1 -1876.423,E2 -1876.423} C_VEL
LIN {X 0,Y 580.773,Z 683.962,A -85,B 0,C 180,E1 -1877.708,E2 -1877.708} C_VEL
LIN {X 0,Y 580.738,Z 697.229,A -85,B 0,C 180,E1 -1878.017,E2 -1878.017} C_VEL
LIN {X 0,Y 580.638,Z 710.5,A -85,B 0,C 180,E1 -1878.48,E2 -1878.48} C_VEL
LIN {X 0,Y 580.564,Z 721.635,A -85,B 0,C 180,E1 -1879.009,E2 -1879.009} C_VEL
LIN {X 0,Y 580.426,Z 733.206,A -85,B 0,C 180,E1 -1879.712,E2 -1879.712} C_VEL
LIN {X 0,Y 580.341,Z 743.601,A -85,B 0,C 180,E1 -1880.503,E2 -1880.503} C_VEL
LIN {X 0,Y 580.271,Z 752.114,A -85,B 0,C 180,E1 -1881.292,E2 -1881.292} C_VEL
LIN {X 0,Y 580.222,Z 759.962,A -85,B 0,C 180,E1 -1882.168,E2 -1882.168} C_VEL
LIN {X 0,Y 580.154,Z 767.651,A -85,B 0,C 180,E1 -1883.222,E2 -1883.222} C_VEL
LIN {X 0,Y 580.139,Z 774.681,A -85,B 0,C 180,E1 -1884.439,E2 -1884.439} C_VEL
LIN {X 0,Y 580.108,Z 779.372,A -85,B 0,C 180,E1 -1885.484,E2 -1885.484} C_VEL
LIN {X 0,Y 580.123,Z 782.957,A -85,B 0,C 180,E1 -1886.527,E2 -1886.527} C_VEL
LIN {X 0,Y 580.043,Z 784.809,A -85,B 0,C 180,E1 -1887.222,E2 -1887.222} C_VEL
LIN {X 0,Y 580.038,Z 786.2,A -85,B 0,C 180,E1 -1887.917,E2 -1887.917} C_VEL
LIN {X 0,Y 580.04,Z 787.784,A -85,B 0,C 180,E1 -1889.306,E2 -1889.306} C_VEL
LIN {X 0,Y 580.037,Z 788,A -85,B 0,C 180,E1 -1890,E2 -1890} C_VEL
LIN {X 0,Y 580.047,Z 787.186,A -85,B 0,C 180,E1 -1891.389,E2 -1891.389} C_VEL
LIN {X 0,Y 580.038,Z 786.201,A -85,B 0,C 180,E1 -1892.083,E2 -1892.083} C_VEL
LIN {X 0,Y 580.043,Z 784.81,A -85,B 0,C 180,E1 -1892.778,E2 -1892.778} C_VEL
LIN {X 0,Y 580.109,Z 781.896,A -85,B 0,C 180,E1 -1893.82,E2 -1893.82} C_VEL
LIN {X 0,Y 580.054,Z 777.95,A -85,B 0,C 180,E1 -1894.865,E2 -1894.865} C_VEL
LIN {X 0,Y 580.139,Z 771.878,A -85,B 0,C 180,E1 -1896.085,E2 -1896.085} C_VEL
LIN {X 0,Y 580.184,Z 765.238,A -85,B 0,C 180,E1 -1897.132,E2 -1897.132} C_VEL
LIN {X 0,Y 580.25,Z 756.992,A -85,B 0,C 180,E1 -1898.182,E2 -1898.182} C_VEL
LIN {X 0,Y 580.308,Z 748.54,A -85,B 0,C 180,E1 -1899.058,E2 -1899.058} C_VEL
LIN {X 0,Y 580.415,Z 738.099,A -85,B 0,C 180,E1 -1899.936,E2 -1899.936} C_VEL
LIN {X 0,Y 580.522,Z 727.761,A -85,B 0,C 180,E1 -1900.639,E2 -1900.639} C_VEL
LIN {X 0,Y 580.597,Z 716.239,A -85,B 0,C 180,E1 -1901.264,E2 -1901.264} C_VEL
LIN {X 0,Y 580.666,Z 703.48,A -85,B 0,C 180,E1 -1901.785,E2 -1901.785} C_VEL
LIN {X 0,Y 580.743,Z 690.447,A -85,B 0,C 180,E1 -1902.16,E2 -1902.16} C_VEL
LIN {X 0,Y 580.833,Z 678.106,A -85,B 0,C 180,E1 -1902.38,E2 -1902.38} C_VEL
LIN {X 0,Y 580.832,Z 578.183,A -85,B 0,C 180,E1 -1903.622,E2 -1903.622} C_VEL
LIN {X 0,Y 580.442,Z 575.272,A -85,B 0,C 180,E1 -1903.679,E2 -1903.679} C_VEL
LIN {X 0,Y 580.603,Z 552.242,A -85,B 0,C 180,E1 -1906.707,E2 -1906.707} C_VEL
LIN {X 0,Y 580.815,Z 531.441,A -85,B 0,C 180,E1 -1909.48,E2 -1909.48} C_VEL
LIN {X 0,Y 581.039,Z 508.571,A -85,B 0,C 180,E1 -1912.583,E2 -1912.583} C_VEL
LIN {X 0,Y 580.953,Z 500.383,A -85,B 0,C 180,E1 -1913.718,E2 -1913.718} C_VEL
LIN {X 0,Y 580.325,Z 497.201,A -85,B 0,C 180,E1 -1914.219,E2 -1914.219} C_VEL
LIN {X 0,Y 580.278,Z 497.207,A -85,B 0,C 180,E1 -1916.623,E2 -1916.623} C_VEL
LIN {X 0,Y 580.301,Z 497.196,A -85,B 0,C 180,E1 -1919.309,E2 -1919.309} C_VEL
LIN {X 0,Y 580.302,Z 497.198,A -85,B 0,C 180,E1 -1922.199,E2 -1922.199} C_VEL
LIN {X 0,Y 580.3,Z 497.205,A -85,B 0,C 180,E1 -1924.695,E2 -1924.695} C_VEL
LIN {X 0,Y 580.3,Z 497.196,A -85,B 0,C 180,E1 -1927.267,E2 -1927.267} C_VEL
LIN {X 0,Y 580.296,Z 497.199,A -85,B 0,C 180,E1 -1930.27,E2 -1930.27} C_VEL
LIN {X 0,Y 580.288,Z 497.206,A -85,B 0,C 180,E1 -1932.704,E2 -1932.704} C_VEL
LIN {X 0,Y 580.27,Z 497.198,A -85,B 0,C 180,E1 -1935.608,E2 -1935.608} C_VEL
LIN {X 0,Y 580.31,Z 497.195,A -85,B 0,C 180,E1 -1938.233,E2 -1938.233} C_VEL
LIN {X 0,Y 580.288,Z 497.203,A -85,B 0,C 180,E1 -1940.965,E2 -1940.965} C_VEL
LIN {X 0,Y 580.292,Z 497.195,A -85,B 0,C 180,E1 -1943.598,E2 -1943.598} C_VEL
LIN {X 0,Y 580.316,Z 497.193,A -85,B 0,C 180,E1 -1946.145,E2 -1946.145} C_VEL
LIN {X 0,Y 580.285,Z 497.203,A -85,B 0,C 180,E1 -1948.615,E2 -1948.615} C_VEL
LIN {X 0,Y 580.291,Z 497.202,A -85,B 0,C 180,E1 -1951.023,E2 -1951.023} C_VEL
LIN {X 0,Y 580.323,Z 497.192,A -85,B 0,C 180,E1 -1953.657,E2 -1953.657} C_VEL
LIN {X 0,Y 580.273,Z 497.2,A -85,B 0,C 180,E1 -1956.441,E2 -1956.441} C_VEL
LIN {X 0,Y 580.276,Z 497.199,A -85,B 0,C 180,E1 -1959.437,E2 -1959.437} C_VEL
LIN {X 0,Y 580.276,Z 497.198,A -85,B 0,C 180,E1 -1961.645,E2 -1961.645} C_VEL
LIN {X 0,Y 580.276,Z 497.197,A -85,B 0,C 180,E1 -1963.825,E2 -1963.825} C_VEL
LIN {X 0,Y 580.317,Z 497.192,A -85,B 0,C 180,E1 -1965.983,E2 -1965.983} C_VEL
LIN {X 0,Y 580.322,Z 497.2,A -85,B 0,C 180,E1 -1968.827,E2 -1968.827} C_VEL
LIN {X 0,Y 580.328,Z 497.192,A -85,B 0,C 180,E1 -1971.644,E2 -1971.644} C_VEL
LIN {X 0,Y 580.324,Z 497.193,A -85,B 0,C 180,E1 -1974.44,E2 -1974.44} C_VEL
LIN {X 0,Y 580.342,Z 497.195,A -85,B 0,C 180,E1 -1977.223,E2 -1977.223} C_VEL
LIN {X 0,Y 580.342,Z 497.189,A -85,B 0,C 180,E1 -1980,E2 -1980} C_VEL
LIN {X 0,Y 580.341,Z 497.195,A -85,B 0,C 180,E1 -1982.776,E2 -1982.776} C_VEL
LIN {X 0,Y 580.328,Z 497.193,A -85,B 0,C 180,E1 -1985.559,E2 -1985.559} C_VEL
LIN {X 0,Y 580.328,Z 497.192,A -85,B 0,C 180,E1 -1988.356,E2 -1988.356} C_VEL
LIN {X 0,Y 580.322,Z 497.2,A -85,B 0,C 180,E1 -1991.208,E2 -1991.208} C_VEL
LIN {X 0,Y 580.317,Z 497.192,A -85,B 0,C 180,E1 -1994.017,E2 -1994.017} C_VEL
LIN {X 0,Y 580.304,Z 497.201,A -85,B 0,C 180,E1 -1996.915,E2 -1996.915} C_VEL
LIN {X 0,Y 580.3,Z 497.196,A -85,B 0,C 180,E1 -1999.822,E2 -1999.822} C_VEL
LIN {X 0,Y 580.278,Z 497.205,A -85,B 0,C 180,E1 -2001.345,E2 -2001.345} C_VEL
LIN {X 0,Y 579.581,Z 497.287,A -85,B 0,C 180,E1 -2001.924,E2 -2001.924} C_VEL
LIN {X 0,Y 576.703,Z 497.648,A -85,B 0,C 180,E1 -2002.863,E2 -2002.863} C_VEL
LIN {X 0,Y 574.307,Z 497.945,A -85,B 0,C 180,E1 -2003.62,E2 -2003.62} C_VEL
LIN {X 0,Y 573.308,Z 498.067,A -85,B 0,C 180,E1 -2004.204,E2 -2004.204} C_VEL
LIN {X 0,Y 573.242,Z 498.075,A -85,B 0,C 180,E1 -2004.401,E2 -2004.401} C_VEL
LIN {X 0,Y 573.258,Z 498.08,A -85,B 0,C 180,E1 -2006.975,E2 -2006.975} C_VEL
LIN {X 0,Y 573.246,Z 498.08,A -85,B 0,C 180,E1 -2009.49,E2 -2009.49} C_VEL
LIN {X 0,Y 573.248,Z 498.075,A -85,B 0,C 180,E1 -2012.23,E2 -2012.23} C_VEL
LIN {X 0,Y 573.3,Z 498.112,A -85,B 0,C 180,E1 -2014.408,E2 -2014.408} C_VEL
LIN {X 0,Y 573.306,Z 509.906,A -85,B 0,C 180,E1 -2016.699,E2 -2016.699} C_VEL
LIN {X 0,Y 573.211,Z 517.854,A -85,B 0,C 180,E1 -2018.226,E2 -2018.226} C_VEL
LIN {X 0,Y 574.068,Z 523.479,A -85,B 0,C 180,E1 -2018.326,E2 -2018.326} C_VEL
LIN {X 0,Y 573.863,Z 624.482,A -85,B 0,C 180,E1 -2019.613,E2 -2019.613} C_VEL
LIN {X 0,Y 573.78,Z 637.852,A -85,B 0,C 180,E1 -2019.933,E2 -2019.933} C_VEL
LIN {X 0,Y 573.681,Z 650.208,A -85,B 0,C 180,E1 -2020.372,E2 -2020.372} C_VEL
LIN {X 0,Y 573.551,Z 662.559,A -85,B 0,C 180,E1 -2020.97,E2 -2020.97} C_VEL
LIN {X 0,Y 573.462,Z 673.609,A -85,B 0,C 180,E1 -2021.659,E2 -2021.659} C_VEL
LIN {X 0,Y 573.283,Z 684.674,A -85,B 0,C 180,E1 -2022.521,E2 -2022.521} C_VEL
LIN {X 0,Y 573.238,Z 694.74,A -85,B 0,C 180,E1 -2023.511,E2 -2023.511} C_VEL
LIN {X 0,Y 573.112,Z 702.945,A -85,B 0,C 180,E1 -2024.503,E2 -2024.503} C_VEL
LIN {X 0,Y 573.085,Z 708.638,A -85,B 0,C 180,E1 -2025.339,E2 -2025.339} C_VEL
LIN {X 0,Y 573.02,Z 714.372,A -85,B 0,C 180,E1 -2026.354,E2 -2026.354} C_VEL
LIN {X 0,Y 573.012,Z 719.803,A -85,B 0,C 180,E1 -2027.58,E2 -2027.58} C_VEL
LIN {X 0,Y 572.967,Z 722.935,A -85,B 0,C 180,E1 -2028.521,E2 -2028.521} C_VEL
LIN {X 0,Y 572.939,Z 725.391,A -85,B 0,C 180,E1 -2029.51,E2 -2029.51} C_VEL
LIN {X 0,Y 572.916,Z 727.151,A -85,B 0,C 180,E1 -2030.608,E2 -2030.608} C_VEL
LIN {X 0,Y 572.922,Z 727.936,A -85,B 0,C 180,E1 -2031.728,E2 -2031.728} C_VEL
LIN {X 0,Y 572.947,Z 727.578,A -85,B 0,C 180,E1 -2033.056,E2 -2033.056} C_VEL
LIN {X 0,Y 572.921,Z 726.352,A -85,B 0,C 180,E1 -2034.058,E2 -2034.058} C_VEL
LIN {X 0,Y 572.981,Z 723.785,A -85,B 0,C 180,E1 -2035.265,E2 -2035.265} C_VEL
LIN {X 0,Y 572.988,Z 719.777,A -85,B 0,C 180,E1 -2036.517,E2 -2036.517} C_VEL
LIN {X 0,Y 573.077,Z 714.047,A -85,B 0,C 180,E1 -2037.799,E2 -2037.799} C_VEL
LIN {X 0,Y 573.115,Z 707.056,A -85,B 0,C 180,E1 -2039.001,E2 -2039.001} C_VEL
LIN {X 0,Y 573.174,Z 699.663,A -85,B 0,C 180,E1 -2040.01,E2 -2040.01} C_VEL
LIN {X 0,Y 573.272,Z 690.337,A -85,B 0,C 180,E1 -2041.038,E2 -2041.038} C_VEL
LIN {X 0,Y 573.377,Z 680.143,A -85,B 0,C 180,E1 -2041.947,E2 -2041.947} C_VEL
LIN {X 0,Y 573.468,Z 668.971,A -85,B 0,C 180,E1 -2042.74,E2 -2042.74} C_VEL
LIN {X 0,Y 573.608,Z 656.558,A -85,B 0,C 180,E1 -2043.432,E2 -2043.432} C_VEL
LIN {X 0,Y 573.719,Z 644.747,A -85,B 0,C 180,E1 -2043.931,E2 -2043.931} C_VEL
LIN {X 0,Y 573.826,Z 631.579,A -85,B 0,C 180,E1 -2044.326,E2 -2044.326} C_VEL
LIN {X 0,Y 573.877,Z 618.491,A -85,B 0,C 180,E1 -2044.572,E2 -2044.572} C_VEL
LIN {X 0,Y 573.95,Z 522.203,A -85,B 0,C 180,E1 -2045.783,E2 -2045.783} C_VEL
LIN {X 0,Y 573.259,Z 517.808,A -85,B 0,C 180,E1 -2045.872,E2 -2045.872} C_VEL
LIN {X 0,Y 573.343,Z 503.223,A -85,B 0,C 180,E1 -2048.685,E2 -2048.685} C_VEL
LIN {X 0,Y 573.269,Z 498.075,A -85,B 0,C 180,E1 -2049.714,E2 -2049.714} C_VEL
LIN {X 0,Y 573.256,Z 498.082,A -85,B 0,C 180,E1 -2052.889,E2 -2052.889} C_VEL
LIN {X 0,Y 573.271,Z 498.07,A -85,B 0,C 180,E1 -2055.807,E2 -2055.807} C_VEL
LIN {X 0,Y 573.26,Z 498.079,A -85,B 0,C 180,E1 -2058.745,E2 -2058.745} C_VEL
LIN {X 0,Y 573.282,Z 498.07,A -85,B 0,C 180,E1 -2061.541,E2 -2061.541} C_VEL
LIN {X 0,Y 573.296,Z 498.069,A -85,B 0,C 180,E1 -2064.372,E2 -2064.372} C_VEL
LIN {X 0,Y 573.312,Z 498.065,A -85,B 0,C 180,E1 -2067.892,E2 -2067.892} C_VEL
LIN {X 0,Y 573.332,Z 498.069,A -85,B 0,C 180,E1 -2070.702,E2 -2070.702} C_VEL
LIN {X 0,Y 573.304,Z 498.074,A -85,B 0,C 180,E1 -2072.811,E2 -2072.811} C_VEL
LIN {X 0,Y 573.295,Z 498.068,A -85,B 0,C 180,E1 -2075.628,E2 -2075.628} C_VEL
LIN {X 0,Y 573.287,Z 498.07,A -85,B 0,C 180,E1 -2078.459,E2 -2078.459} C_VEL
LIN {X 0,Y 573.269,Z 498.074,A -85,B 0,C 180,E1 -2081.312,E2 -2081.312} C_VEL
LIN {X 0,Y 573.271,Z 498.07,A -85,B 0,C 180,E1 -2084.193,E2 -2084.193} C_VEL
LIN {X 0,Y 573.256,Z 498.08,A -85,B 0,C 180,E1 -2087.111,E2 -2087.111} C_VEL
LIN {X 0,Y 573.25,Z 498.072,A -85,B 0,C 180,E1 -2090.076,E2 -2090.076} C_VEL
LIN {X 0,Y 573.23,Z 498.083,A -85,B 0,C 180,E1 -2093.099,E2 -2093.099} C_VEL
LIN {X 0,Y 573.25,Z 498.076,A -85,B 0,C 180,E1 -2095.41,E2 -2095.41} C_VEL
LIN {X 0,Y 573.259,Z 498.071,A -85,B 0,C 180,E1 -2098.031,E2 -2098.031} C_VEL
LIN {X 0,Y 573.241,Z 498.082,A -85,B 0,C 180,E1 -2100.885,E2 -2100.885} C_VEL
LIN {X 0,Y 573.256,Z 498.074,A -85,B 0,C 180,E1 -2103.524,E2 -2103.524} C_VEL
LIN {X 0,Y 573.255,Z 498.072,A -85,B 0,C 180,E1 -2106.048,E2 -2106.048} C_VEL
LIN {X 0,Y 573.245,Z 498.078,A -85,B 0,C 180,E1 -2108.7,E2 -2108.7} C_VEL
LIN {X 0,Y 573.259,Z 498.073,A -85,B 0,C 180,E1 -2111.597,E2 -2111.597} C_VEL
LIN {X 0,Y 573.231,Z 498.075,A -85,B 0,C 180,E1 -2114.333,E2 -2114.333} C_VEL
LIN {X 0,Y 573.235,Z 498.08,A -85,B 0,C 180,E1 -2117.358,E2 -2117.358} C_VEL
LIN {X 0,Y 573.242,Z 498.074,A -85,B 0,C 180,E1 -2120.393,E2 -2120.393} C_VEL
LIN {X 0,Y 573.248,Z 498.083,A -85,B 0,C 180,E1 -2123.078,E2 -2123.078} C_VEL
LIN {X 0,Y 573.268,Z 498.072,A -85,B 0,C 180,E1 -2125.672,E2 -2125.672} C_VEL
LIN {X 0,Y 573.241,Z 498.073,A -85,B 0,C 180,E1 -2128.185,E2 -2128.185} C_VEL
LIN {X 0,Y 573.263,Z 498.074,A -85,B 0,C 180,E1 -2130.635,E2 -2130.635} C_VEL
LIN {X 0,Y 573.264,Z 498.075,A -85,B 0,C 180,E1 -2133.499,E2 -2133.499} C_VEL
LIN {X 0,Y 573.224,Z 498.076,A -85,B 0,C 180,E1 -2136.135,E2 -2136.135} C_VEL
LIN {X 0,Y 573.252,Z 498.082,A -85,B 0,C 180,E1 -2139.174,E2 -2139.174} C_VEL
LIN {X 0,Y 573.231,Z 498.08,A -85,B 0,C 180,E1 -2141.412,E2 -2141.412} C_VEL
LIN {X 0,Y 573.25,Z 498.075,A -85,B 0,C 180,E1 -2143.622,E2 -2143.622} C_VEL
LIN {X 0,Y 573.23,Z 498.076,A -85,B 0,C 180,E1 -2146.53,E2 -2146.53} C_VEL
LIN {X 0,Y 573.272,Z 498.073,A -85,B 0,C 180,E1 -2148.734,E2 -2148.734} C_VEL
LIN {X 0,Y 573.299,Z 498.071,A -85,B 0,C 180,E1 -2151.541,E2 -2151.541} C_VEL
LIN {X 0,Y 573.291,Z 498.067,A -85,B 0,C 180,E1 -2154.372,E2 -2154.372} C_VEL
LIN {X 0,Y 573.3,Z 498.067,A -85,B 0,C 180,E1 -2157.893,E2 -2157.893} C_VEL
LIN {X 0,Y 573.33,Z 498.065,A -85,B 0,C 180,E1 -2160.703,E2 -2160.703} C_VEL
LIN {X 0,Y 573.24,Z 498.079,A -85,B 0,C 180,E1 -2163.515,E2 -2163.515} C_VEL
LIN {X 0,Y 573.296,Z 498.07,A -85,B 0,C 180,E1 -2165.628,E2 -2165.628} C_VEL
LIN {X 0,Y 573.301,Z 498.066,A -85,B 0,C 180,E1 -2168.46,E2 -2168.46} C_VEL
LIN {X 0,Y 573.29,Z 498.077,A -85,B 0,C 180,E1 -2171.312,E2 -2171.312} C_VEL
LIN {X 0,Y 573.272,Z 498.07,A -85,B 0,C 180,E1 -2174.425,E2 -2174.425} C_VEL
LIN {X 0,Y 573.252,Z 498.08,A -85,B 0,C 180,E1 -2177.112,E2 -2177.112} C_VEL
LIN {X 0,Y 573.25,Z 498.073,A -85,B 0,C 180,E1 -2180.077,E2 -2180.077} C_VEL
LIN {X 0,Y 573.232,Z 498.075,A -85,B 0,C 180,E1 -2182.338,E2 -2182.338} C_VEL
LIN {X 0,Y 573.251,Z 498.081,A -85,B 0,C 180,E1 -2185.411,E2 -2185.411} C_VEL
LIN {X 0,Y 573.258,Z 498.072,A -85,B 0,C 180,E1 -2188.033,E2 -2188.033} C_VEL
LIN {X 0,Y 573.238,Z 498.077,A -85,B 0,C 180,E1 -2190.886,E2 -2190.886} C_VEL
LIN {X 0,Y 573.282,Z 498.075,A -85,B 0,C 180,E1 -2193.529,E2 -2193.529} C_VEL
LIN {X 0,Y 573.256,Z 498.072,A -85,B 0,C 180,E1 -2196.049,E2 -2196.049} C_VEL
LIN {X 0,Y 573.246,Z 498.074,A -85,B 0,C 180,E1 -2198.702,E2 -2198.702} C_VEL
LIN {X 0,Y 573.25,Z 498.078,A -85,B 0,C 180,E1 -2201.597,E2 -2201.597} C_VEL
LIN {X 0,Y 573.235,Z 498.074,A -85,B 0,C 180,E1 -2204.334,E2 -2204.334} C_VEL
LIN {X 0,Y 573.248,Z 498.083,A -85,B 0,C 180,E1 -2207.358,E2 -2207.358} C_VEL
LIN {X 0,Y 573.246,Z 498.073,A -85,B 0,C 180,E1 -2210.394,E2 -2210.394} C_VEL
LIN {X 0,Y 573.254,Z 498.077,A -85,B 0,C 180,E1 -2213.079,E2 -2213.079} C_VEL
LIN {X 0,Y 573.268,Z 498.076,A -85,B 0,C 180,E1 -2215.672,E2 -2215.672} C_VEL
LIN {X 0,Y 573.249,Z 498.074,A -85,B 0,C 180,E1 -2218.186,E2 -2218.186} C_VEL
LIN {X 0,Y 573.264,Z 498.072,A -85,B 0,C 180,E1 -2220.635,E2 -2220.635} C_VEL
LIN {X 0,Y 573.252,Z 498.078,A -85,B 0,C 180,E1 -2223.025,E2 -2223.025} C_VEL
LIN {X 0,Y 573.3,Z 498.165,A -85,B 0,C 180,E1 -2225.633,E2 -2225.633} C_VEL
LIN {X 0,Y 574.199,Z 504.007,A -85,B 0,C 180,E1 -2226.495,E2 -2226.495} C_VEL
LIN {X 0,Y 573.949,Z 523.583,A -85,B 0,C 180,E1 -2229.201,E2 -2229.201} C_VEL
LIN {X 0,Y 573.75,Z 542.689,A -85,B 0,C 180,E1 -2231.799,E2 -2231.799} C_VEL
LIN {X 0,Y 573.483,Z 564.525,A -85,B 0,C 180,E1 -2234.724,E2 -2234.724} C_VEL
LIN {X 0,Y 573.44,Z 575.357,A -85,B 0,C 180,E1 -2236.162,E2 -2236.162} C_VEL
LIN {X 0,Y 574.084,Z 581.535,A -85,B 0,C 180,E1 -2236.257,E2 -2236.257} C_VEL
LIN {X 0,Y 573.837,Z 683.962,A -85,B 0,C 180,E1 -2237.557,E2 -2237.557} C_VEL
LIN {X 0,Y 573.796,Z 697.229,A -85,B 0,C 180,E1 -2237.87,E2 -2237.87} C_VEL
LIN {X 0,Y 573.689,Z 710.501,A -85,B 0,C 180,E1 -2238.339,E2 -2238.339} C_VEL
LIN {X 0,Y 573.576,Z 721.711,A -85,B 0,C 180,E1 -2238.878,E2 -2238.878} C_VEL
LIN {X 0,Y 573.437,Z 733.207,A -85,B 0,C 180,E1 -2239.585,E2 -2239.585} C_VEL
LIN {X 0,Y 573.326,Z 743.602,A -85,B 0,C 180,E1 -2240.386,E2 -2240.386} C_VEL
LIN {X 0,Y 573.241,Z 752.115,A -85,B 0,C 180,E1 -2241.185,E2 -2241.185} C_VEL
LIN {X 0,Y 573.161,Z 759.962,A -85,B 0,C 180,E1 -2242.071,E2 -2242.071} C_VEL
LIN {X 0,Y 573.073,Z 767.956,A -85,B 0,C 180,E1 -2243.186,E2 -2243.186} C_VEL
LIN {X 0,Y 573.07,Z 774.681,A -85,B 0,C 180,E1 -2244.37,E2 -2244.37} C_VEL
LIN {X 0,Y 573.029,Z 779.372,A -85,B 0,C 180,E1 -2245.428,E2 -2245.428} C_VEL
LIN {X 0,Y 573.022,Z 782.957,A -85,B 0,C 180,E1 -2246.484,E2 -2246.484} C_VEL
LIN {X 0,Y 572.959,Z 784.808,A -85,B 0,C 180,E1 -2247.188,E2 -2247.188} C_VEL
LIN {X 0,Y 572.937,Z 786.199,A -85,B 0,C 180,E1 -2247.891,E2 -2247.891} C_VEL
LIN {X 0,Y 572.941,Z 787.785,A -85,B 0,C 180,E1 -2249.297,E2 -2249.297} C_VEL
LIN {X 0,Y 572.938,Z 788,A -85,B 0,C 180,E1 -2250,E2 -2250} C_VEL
LIN {X 0,Y 572.946,Z 787.186,A -85,B 0,C 180,E1 -2251.406,E2 -2251.406} C_VEL
LIN {X 0,Y 572.937,Z 786.2,A -85,B 0,C 180,E1 -2252.109,E2 -2252.109} C_VEL
LIN {X 0,Y 572.959,Z 784.81,A -85,B 0,C 180,E1 -2252.812,E2 -2252.812} C_VEL
LIN {X 0,Y 573.014,Z 781.896,A -85,B 0,C 180,E1 -2253.868,E2 -2253.868} C_VEL
LIN {X 0,Y 572.963,Z 777.95,A -85,B 0,C 180,E1 -2254.925,E2 -2254.925} C_VEL
LIN {X 0,Y 573.064,Z 771.878,A -85,B 0,C 180,E1 -2256.16,E2 -2256.16} C_VEL
LIN {X 0,Y 573.119,Z 765.239,A -85,B 0,C 180,E1 -2257.221,E2 -2257.221} C_VEL
LIN {X 0,Y 573.201,Z 756.992,A -85,B 0,C 180,E1 -2258.283,E2 -2258.283} C_VEL
LIN {X 0,Y 573.286,Z 748.541,A -85,B 0,C 180,E1 -2259.17,E2 -2259.17} C_VEL
LIN {X 0,Y 573.42,Z 738.1,A -85,B 0,C 180,E1 -2260.058,E2 -2260.058} C_VEL
LIN {X 0,Y 573.546,Z 726.358,A -85,B 0,C 180,E1 -2260.857,E2 -2260.857} C_VEL
LIN {X 0,Y 573.653,Z 715.287,A -85,B 0,C 180,E1 -2261.447,E2 -2261.447} C_VEL
LIN {X 0,Y 573.749,Z 702.182,A -85,B 0,C 180,E1 -2261.974,E2 -2261.974} C_VEL
LIN {X 0,Y 573.834,Z 689.532,A -85,B 0,C 180,E1 -2262.331,E2 -2262.331} C_VEL
LIN {X 0,Y 573.936,Z 676.334,A -85,B 0,C 180,E1 -2262.553,E2 -2262.553} C_VEL
LIN {X 0,Y 573.927,Z 578.854,A -85,B 0,C 180,E1 -2263.781,E2 -2263.781} C_VEL
LIN {X 0,Y 573.447,Z 575.272,A -85,B 0,C 180,E1 -2263.849,E2 -2263.849} C_VEL
LIN {X 0,Y 573.633,Z 552.252,A -85,B 0,C 180,E1 -2266.915,E2 -2266.915} C_VEL
LIN {X 0,Y 573.87,Z 531.771,A -85,B 0,C 180,E1 -2269.681,E2 -2269.681} C_VEL
LIN {X 0,Y 574.139,Z 509.936,A -85,B 0,C 180,E1 -2272.68,E2 -2272.68} C_VEL
LIN {X 0,Y 574.18,Z 502.776,A -85,B 0,C 180,E1 -2273.679,E2 -2273.679} C_VEL
LIN {X 0,Y 573.289,Z 498.078,A -85,B 0,C 180,E1 -2274.391,E2 -2274.391} C_VEL
LIN {X 0,Y 573.252,Z 498.078,A -85,B 0,C 180,E1 -2276.975,E2 -2276.975} C_VEL
LIN {X 0,Y 573.247,Z 498.074,A -85,B 0,C 180,E1 -2279.487,E2 -2279.487} C_VEL
LIN {X 0,Y 573.255,Z 498.077,A -85,B 0,C 180,E1 -2282.228,E2 -2282.228} C_VEL
LIN {X 0,Y 573.25,Z 498.082,A -85,B 0,C 180,E1 -2284.773,E2 -2284.773} C_VEL
LIN {X 0,Y 573.254,Z 498.075,A -85,B 0,C 180,E1 -2287.165,E2 -2287.165} C_VEL
LIN {X 0,Y 573.246,Z 498.073,A -85,B 0,C 180,E1 -2289.606,E2 -2289.606} C_VEL
LIN {X 0,Y 573.248,Z 498.083,A -85,B 0,C 180,E1 -2292.642,E2 -2292.642} C_VEL
LIN {X 0,Y 573.235,Z 498.074,A -85,B 0,C 180,E1 -2295.666,E2 -2295.666} C_VEL
LIN {X 0,Y 573.241,Z 498.08,A -85,B 0,C 180,E1 -2298.543,E2 -2298.543} C_VEL
LIN {X 0,Y 573.246,Z 498.075,A -85,B 0,C 180,E1 -2301.298,E2 -2301.298} C_VEL
LIN {X 0,Y 573.26,Z 498.072,A -85,B 0,C 180,E1 -2304.01,E2 -2304.01} C_VEL
LIN {X 0,Y 573.279,Z 498.074,A -85,B 0,C 180,E1 -2306.518,E2 -2306.518} C_VEL
